FUNCTION_BLOCK FB_Lifetime_Predictor
  VAR_INPUT
    VI_Runtime_Hours : UDINT;
    VI_Start_Count : UDINT;
    VI_Nominal_Life : UDINT := 10000;
  END_VAR
  VAR_OUTPUT
    VO_Remaining_Percent : BYTE;
    VO_Maintenance_Req : BOOL;
  END_VAR

            // Упрощенная модель износа
IF VI_Nominal_Life > 0 THEN
    VO_Remaining_Percent := TO_BYTE(100 - (VI_Runtime_Hours * 100 / VI_Nominal_Life));
ELSE
    VO_Remaining_Percent := 0;
END_IF;

VO_Maintenance_Req := (VO_Remaining_Percent < 10);
          
END_FUNCTION_BLOCK

FUNCTION_BLOCK FB_System_Alarm_Orchestrator
  VAR_INPUT
    VI_First_Fault_Active : BOOL;
    VI_First_Fault_Type : INT;
    VI_First_Fault_Source : INT;
  END_VAR
  VAR
    fbAlarmManager : FB_Alarm_Manager;
  END_VAR

            // ==============================================================================
// System alarm orchestrator helper
//
// Internal helper for PRG_System.
// Owns FB_Alarm_Manager call and alarm output projection.
// ==============================================================================



fbAlarmManager(
    VI_System_Time_MS := GVL_STATUS.G_System_Time_MS,
    VI_IsActivePLC := GVL_STATUS.G_Is_Active_PLC,
    VI_Gas_Alarm := GVL_HEALTH_BRIDGE.G_Gas_Detected OR GVL_HEALTH_BRIDGE.G_CO_Alarm_Level,
    VI_Fire_Alarm := GVL_HEALTH_BRIDGE.G_Smoke_Detected,
    VI_Flood_Alarm := GVL_HEALTH_BRIDGE.G_Leak_Detected,
    VI_Security_Alarm := GVL_ALARM.G_Security_Alarm,
    VI_First_Fault_Active := VI_First_Fault_Active,
    VI_First_Fault_Type := VI_First_Fault_Type,
    VI_First_Fault_Source := VI_First_Fault_Source,
    VI_Boiler_Errors := GVL_STATE.G_Boiler_Error,
    VI_Security_Msg := GVL_STATUS.G_Security_Status_Msg,
    VI_Acknowledge_All := GVL_CONFIG.G_HMI_Ack_Alarms OR GVL_COMMAND.G_Reset_Errors,
    VI_Mute_Siren := GVL_CONFIG.G_HMI_Mute_Alarm,
    VIO_Next_Alarm_ID := GVL_ALARM.G_Next_Alarm_ID,
    VO_Global_Critical => GVL_ALARM.G_Global_Critical,
    VO_Global_Warning => GVL_ALARM.G_Global_Warning,
    VO_Siren_Active => GVL_ALARM.G_Global_Siren,
    VO_Active_Count => GVL_ALARM.G_Active_Alarm_Count,
    VO_Unacked_Count => GVL_ALARM.G_Unacked_Alarm_Count,
    VO_Event_Pulse => GVL_STATUS.G_Diagnostics.Alarm_Event_Pulse,
    VO_Event_Code => GVL_STATUS.G_Diagnostics.Alarm_Event_Code,
    VO_Event_Value => GVL_STATUS.G_Diagnostics.Alarm_Event_Value,
    VO_Alarm_List => GVL_ALARM.G_Alarm_List
);

// >>> BULK_SYNC_ANCHOR: FB_System_Alarm_Orchestrator <<<
          
END_FUNCTION_BLOCK

FUNCTION_BLOCK FB_Heating_Runtime_Timeline_Observer
  VAR_INPUT
    VI_Enable : BOOL;
    VI_Frame : ST_Heating_Runtime_Execution_Frame;
  END_VAR
  VAR_IN_OUT
    VIO_Timeline : ST_Heating_Runtime_Execution_Timeline;
  END_VAR
  VAR
    L_Index : UINT;
  END_VAR

            // ==============================================================================
// Heating runtime timeline observer
// Read-only deterministic execution timeline layer.
// ==============================================================================



IF NOT VI_Enable THEN
    RETURN;
END_IF;

// ======================================================
// SAFE INDEX NORMALIZATION
// ======================================================
IF (VIO_Timeline.Write_Index < 1) OR
   (VIO_Timeline.Write_Index >= 64) THEN

    L_Index := 1;

    IF VIO_Timeline.Write_Index >= 64 THEN
        VIO_Timeline.Timeline_Overflow := TRUE;
    END_IF;

ELSE
    L_Index := VIO_Timeline.Write_Index + 1;
END_IF;

// ======================================================
// FRAME STORAGE
// ======================================================
VIO_Timeline.Frames[L_Index] := VI_Frame;
VIO_Timeline.Write_Index := L_Index;

IF VIO_Timeline.Frame_Count < 64 THEN
    VIO_Timeline.Frame_Count :=
        VIO_Timeline.Frame_Count + 1;
END_IF;

// ======================================================
// TELEMETRY UPDATE
// ======================================================
VIO_Timeline.Sequencing_Valid :=
    VI_Frame.Sequencing_Valid;

VIO_Timeline.Ownership_Valid :=
    VI_Frame.Ownership_Valid;

VIO_Timeline.Synchronization_Valid :=
    VI_Frame.Synchronization_Valid;

VIO_Timeline.Runtime_Jitter_Detected :=
    VI_Frame.Runtime_Jitter_Detected;

VIO_Timeline.Runtime_Latency_Detected :=
    VI_Frame.Runtime_Latency_Detected;

VIO_Timeline.Runtime_Degraded :=
    VI_Frame.Runtime_Degraded;

VIO_Timeline.Status_Code := VI_Frame.Status_Code;
VIO_Timeline.Status_Text := VI_Frame.Status_Text;

// >>> BULK_SYNC_ANCHOR: FB_Heating_Runtime_Timeline_Observer <<<
          
END_FUNCTION_BLOCK

FUNCTION_BLOCK FB_Behavior_Adapt
  VAR_INPUT
    iScenario : E_System_Reason_Code;
    iSuccess : BOOL;
    iMeasuredValue : REAL;
    iZone : INT;
    iConfidence : REAL;
  END_VAR
  VAR
    L_Stats : ST_Scenario_Stats;
    L_Zone : ST_Zone_Adapt_State;
    L_Adjustment : REAL;
    L_Decay : REAL;
    idx : INT;
  END_VAR

            IF NOT GVL_BEHAVIOR_ADAPT.G_Adapt_Enabled THEN RETURN; END_IF;

idx := USINT_TO_INT(iScenario);

L_Stats := GVL_BEHAVIOR_ADAPT.G_Scenario_Stats[idx];
L_Stats.Activations := L_Stats.Activations + 1;

IF iSuccess THEN
    L_Stats.Success_Count := L_Stats.Success_Count + 1;
ELSE
    L_Stats.Failure_Count := L_Stats.Failure_Count + 1;
END_IF;

IF L_Stats.Activations > 0 THEN
    L_Stats.Success_Rate := UDINT_TO_REAL(L_Stats.Success_Count) / UDINT_TO_REAL(L_Stats.Activations);
END_IF;

IF (iScenario = REASON_SCENARIO_VENT_BOOST) AND (iZone >= 1) AND (iZone <= GVL_CONSTANTS.C_MAX_ZONES) THEN

    L_Zone := GVL_BEHAVIOR_ADAPT.G_VentBoost_Zone_Adapt[iZone];

    IF L_Zone.Zone_Weight = 0.0 THEN
        L_Zone.Zone_Weight := GVL_BEHAVIOR_ADAPT.G_Adapt_Default_Zone_Weight;
    END_IF;

    L_Decay := GVL_BEHAVIOR_ADAPT.G_Decay_Factor;
    L_Zone.Zone_Weight := L_Zone.Zone_Weight * L_Decay;
    L_Zone.Confidence := L_Zone.Confidence * L_Decay;

    L_Zone.Activations := L_Zone.Activations + 1;

    IF iSuccess THEN
        L_Zone.Success_Count := L_Zone.Success_Count + 1;
    ELSE
        L_Zone.Failure_Count := L_Zone.Failure_Count + 1;
    END_IF;

    IF L_Zone.Activations > 0 THEN
        L_Zone.Success_Rate := UDINT_TO_REAL(L_Zone.Success_Count) / UDINT_TO_REAL(L_Zone.Activations);
    END_IF;

    IF iConfidence >= GVL_BEHAVIOR_ADAPT.G_Adapt_Min_Confidence THEN
        L_Zone.Confidence := L_Zone.Confidence +
            (iConfidence - L_Zone.Confidence) * GVL_BEHAVIOR_ADAPT.G_Confidence_Learning_Rate;
    END_IF;

    IF (GVL_BEHAVIOR_ADAPT.G_Adapt_Update_Threshold > 0) AND
       ((L_Zone.Activations MOD INT_TO_UDINT(GVL_BEHAVIOR_ADAPT.G_Adapt_Update_Threshold)) = 0) THEN

        L_Adjustment :=
            (L_Zone.Success_Rate - 0.5)
            * GVL_BEHAVIOR_ADAPT.G_Adapt_Learning_Rate
            * L_Zone.Confidence;

        L_Zone.Zone_Weight := LIMIT(0.5, L_Zone.Zone_Weight + L_Adjustment, 2.0);

    END_IF;

    L_Zone.Last_Update_MS := GVL_TIME_SERVICE.G_Now_MS;

    GVL_BEHAVIOR_ADAPT.G_VentBoost_Zone_Adapt[iZone] := L_Zone;

END_IF;

GVL_BEHAVIOR_ADAPT.G_Scenario_Stats[idx] := L_Stats;
          
END_FUNCTION_BLOCK

FUNCTION_BLOCK FB_Heating_Optimizer
  VAR
    L_i : INT;
    L_Load : REAL;
    L_Total_Demand : REAL;
  END_VAR

            // ==============================================================================
// Ownership note
// ------------------------------------------------------------------------------
// This block calculates optimization diagnostics only.
// It does NOT modify thermal demand.
//
// Thermal demand ownership remains in:
// FB_Heating_Thermal_Model.
// ==============================================================================

L_Total_Demand := 0.0;

// Aggregate thermal load estimate.
FOR L_i := 1 TO GVL_CONSTANTS.C_MAX_ZONES DO
    L_Total_Demand := L_Total_Demand + ABS(GVL_HEATING_POLICY.G_Zone_Thermal_Demand[L_i]);
END_FOR;

GVL_HEATING_POLICY.G_Optimization_Load_Index := L_Total_Demand;
GVL_HEATING_POLICY.G_Optimization_Energy_Saving_Active := FALSE;

// Zone optimization diagnostics.
FOR L_i := 1 TO GVL_CONSTANTS.C_MAX_ZONES DO

    IF L_Total_Demand > 0.01 THEN
        L_Load := ABS(GVL_HEATING_POLICY.G_Zone_Thermal_Demand[L_i]) / L_Total_Demand;
    ELSE
        L_Load := 0.0;
    END_IF;

    GVL_HEATING_POLICY.G_Zone_Optimization_Score[L_i] :=
        L_Load +
        ((1.0 - GVL_HEATING_POLICY.G_Zone_Thermal_Model_Confidence[L_i]) * 0.2);

    // Advisory energy-saving indication only.
    IF L_Total_Demand > 5.0 THEN
        GVL_HEATING_POLICY.G_Optimization_Energy_Saving_Active := TRUE;
    END_IF;

END_FOR;
          
END_FUNCTION_BLOCK

FUNCTION_BLOCK FB_System_Timebase
  VAR
    L_Time_Diff : UDINT;
  END_VAR

            // ==============================================================================
// System timebase helper
//
// Internal helper for PRG_System.
// Owns PLC runtime clock projection into GVL_STATUS:
// - monotonic system milliseconds
// - time-of-day milliseconds
// - day of week / day of year rollover
// - TOD representation
// ==============================================================================



GVL_STATUS.G_System_Time_MS := TIME_TO_UDINT(TIME());

L_Time_Diff := SEL(
    GVL_STATUS.G_System_Time_MS >= GVL_STATUS.G_Last_System_Time_MS,
    GVL_STATUS.G_System_Time_MS - GVL_STATUS.G_Last_System_Time_MS,
    (4294967295 - GVL_STATUS.G_Last_System_Time_MS) + GVL_STATUS.G_System_Time_MS + 1
);

GVL_STATUS.G_Time_Of_Day_MS := (GVL_STATUS.G_Time_Of_Day_MS + L_Time_Diff) MOD 86400000;

IF GVL_STATUS.G_Time_Of_Day_MS < L_Time_Diff THEN
    GVL_STATUS.G_Current_Day := (GVL_STATUS.G_Current_Day MOD 7) + 1;
    GVL_STATUS.G_Day_Of_Year := (GVL_STATUS.G_Day_Of_Year MOD 365) + 1;
END_IF;

GVL_STATUS.G_Last_System_Time_MS := GVL_STATUS.G_System_Time_MS;
GVL_STATUS.G_Current_TOD := UDINT_TO_TOD(GVL_STATUS.G_Time_Of_Day_MS);

// >>> BULK_SYNC_ANCHOR: FB_System_Timebase <<<
          
END_FUNCTION_BLOCK

FUNCTION_BLOCK FB_Redundancy_Manager
  VAR_INPUT
    VI_System_Time_MS : UDINT;
    VI_Local_PLC_ID : BYTE;
    VI_Remote_Pulse : BOOL;
    VI_Remote_Is_Active : BOOL;
    VI_Gateway_Ping_OK : BOOL;
    VI_Remote_State : ST_System_State_Snapshot;
    VI_Local_State : ST_System_State_Snapshot;
  END_VAR
  VAR_OUTPUT
    VO_Local_Role : E_PLC_ROLE;
    VO_Local_Pulse : BOOL;
    VO_Sync_Data_Req : BOOL;
    VO_Status_Msg : STRING(200);
    VO_Synced_State : ST_System_State_Snapshot;
    VO_State_Updated : BOOL;
  END_VAR
  VAR
    L_Heartbeat : FB_PLC_Heartbeat;
    L_Pulse_Timer : FB_System_Timer;
    L_Pulse_State : BOOL;
    L_Prev_Role : E_PLC_ROLE;
    L_State_Replicator : FB_State_Replication;
  END_VAR

            // 1. Генерация собственного пульса (меандр 100 мс)
L_Pulse_Timer(IN := NOT L_Pulse_Timer.Q, PT := T#100ms, VI_System_Time_MS := VI_System_Time_MS);
IF L_Pulse_Timer.Q THEN
    L_Pulse_State := NOT L_Pulse_State;
END_IF;
VO_Local_Pulse := L_Pulse_State;

// 2. Определение роли через Heartbeat
L_Heartbeat(
    VI_Local_ID := VI_Local_PLC_ID,
    VI_System_Time := VI_System_Time_MS,
    VI_Remote_Pulse := VI_Remote_Pulse,
    VI_Remote_Is_Active := VI_Remote_Is_Active,
    VI_Gateway_Ping_OK := VI_Gateway_Ping_OK
);

IF L_Heartbeat.VO_Is_Active THEN
    VO_Local_Role := E_PLC_ROLE.ROLE_ACTIVE;
    VO_Status_Msg := 'ПЛК АКТИВЕН (ВЕДУЩИЙ)';
ELSE
    VO_Local_Role := E_PLC_ROLE.ROLE_STANDBY;
    VO_Status_Msg := 'ПЛК В РЕЗЕРВЕ (ВЕДОМЫЙ)';
END_IF;

// 3. Запрос на синхронизацию при переходе в ACTIVE
IF VO_Local_Role = E_PLC_ROLE.ROLE_ACTIVE AND L_Prev_Role = E_PLC_ROLE.ROLE_STANDBY THEN
    VO_Sync_Data_Req := TRUE;
ELSE
    VO_Sync_Data_Req := FALSE;
END_IF;

L_State_Replicator(
    VI_Local_Role := VO_Local_Role,
    VI_Sync_Req := VO_Sync_Data_Req,
    VI_Local_State := VI_Local_State,
    VI_Remote_State := VI_Remote_State,
    VI_System_Time_MS := VI_System_Time_MS
);
VO_Synced_State := L_State_Replicator.VO_Synced_State;
VO_State_Updated := L_State_Replicator.VO_State_Updated;

L_Prev_Role := VO_Local_Role;
// >>> BULK_SYNC_ANCHOR: FB_Redundancy_Manager <<<
          
END_FUNCTION_BLOCK

FUNCTION_BLOCK FB_System_Redundancy_Orchestrator
  VAR_IN_OUT
    VIO_Local_State : ST_System_State_Snapshot;
    VIO_Remote_State : ST_System_State_Snapshot;
  END_VAR
  VAR
    fbRedundancy : FB_Redundancy_Manager;
  END_VAR

            // ==============================================================================
// System redundancy orchestrator helper
//
// Internal helper for PRG_System.
// Owns PLC role calculation, heartbeat output projection, and synced-state apply.
// ==============================================================================



// Build local state snapshot for replication.
VIO_Local_State.System_Time_MS := GVL_STATUS.G_System_Time_MS;
VIO_Local_State.Current_Scenario := GVL_STATUS.G_Current_Scenario;
VIO_Local_State.Security_Armed := GVL_ALARM.G_Security_Armed;
VIO_Local_State.Active_Alarms := GVL_ALARM.G_Active_Alarm_Count;
VIO_Local_State.Zone_Valves := GVL_STATE.G_Zone_Valves;
VIO_Local_State.Manifold_Pumps := GVL_STATE.G_Manifold_Pumps;
VIO_Local_State.Lighting_States := GVL_STATE.G_Lighting_Levels;
VIO_Local_State.Blinds_Positions := GVL_STATE.G_Blinds_Positions;
VIO_Local_State.Socket_States := GVL_STATE.G_Socket_States;
VIO_Local_State.Gas_Valve_Closed := GVL_COMMAND.G_Gas_Valve_Close;
VIO_Local_State.Water_Valves_Closed := GVL_COMMAND.G_Close_Valve_36;
VIO_Local_State.Version := VIO_Local_State.Version + 1;

fbRedundancy(
    VI_System_Time_MS := GVL_STATUS.G_System_Time_MS,
    VI_Local_PLC_ID := GVL_STATUS.G_PLC_ID,
    VI_Remote_Pulse := GVL_IO.DI_Partner_Pulse,
    VI_Remote_Is_Active := GVL_IO.DI_Partner_Active,
    VI_Gateway_Ping_OK := GVL_GATEWAY.G_Gateway_Ping_OK,
    VI_Local_State := VIO_Local_State,
    VI_Remote_State := VIO_Remote_State
);

GVL_STATUS.G_Is_Active_PLC := (fbRedundancy.VO_Local_Role = E_PLC_ROLE.ROLE_ACTIVE);
GVL_IO.DO_Heartbeat_Pulse := fbRedundancy.VO_Local_Pulse;
GVL_IO.DO_Active_Status := GVL_STATUS.G_Is_Active_PLC;

IF fbRedundancy.VO_State_Updated THEN
    GVL_STATUS.G_Current_Scenario := fbRedundancy.VO_Synced_State.Current_Scenario;
    GVL_ALARM.G_Security_Armed := fbRedundancy.VO_Synced_State.Security_Armed;
    GVL_STATE.G_Zone_Valves := fbRedundancy.VO_Synced_State.Zone_Valves;
    GVL_STATE.G_Manifold_Pumps := fbRedundancy.VO_Synced_State.Manifold_Pumps;
    GVL_STATE.G_Lighting_Levels := fbRedundancy.VO_Synced_State.Lighting_States;
    GVL_STATE.G_Blinds_Positions := fbRedundancy.VO_Synced_State.Blinds_Positions;
    GVL_STATE.G_Socket_States := fbRedundancy.VO_Synced_State.Socket_States;
    GVL_COMMAND.G_Gas_Valve_Close := fbRedundancy.VO_Synced_State.Gas_Valve_Closed;
    GVL_COMMAND.G_Close_Valve_36 := fbRedundancy.VO_Synced_State.Water_Valves_Closed;
    VIO_Local_State.Version := fbRedundancy.VO_Synced_State.Version;
END_IF;

// >>> BULK_SYNC_ANCHOR: FB_System_Redundancy_Orchestrator <<<
          
END_FUNCTION_BLOCK

FUNCTION_BLOCK FB_Heating_Boiler_Control
  VAR_INPUT
    VI_System_Time_MS : UDINT;
    VI_IsActivePLC : BOOL;
    VI_DHW_Heating_Demand : BOOL;
    VI_DHW_Target_Temp : REAL;
    VI_Target_Supply_Temp : REAL;
    VI_Freeze_Mode_Active : BOOL;
    VI_Policy_Degraded : BOOL;
    VI_Manifold_Pumps : ARRAY[1..GVL_CONSTANTS.C_MAX_MANIFOLDS] OF BOOL;
    VI_Manifold_Valves : ARRAY[1..GVL_CONSTANTS.C_MAX_MANIFOLDS] OF REAL;
    VI_Boiler_Flame_Status : ARRAY[1..GVL_CONSTANTS.C_MAX_BOILERS] OF BOOL;
    VI_Boiler_Error_Status : ARRAY[1..GVL_CONSTANTS.C_MAX_BOILERS] OF BOOL;
    VI_Boiler_OT_Online : ARRAY[1..GVL_CONSTANTS.C_MAX_BOILERS] OF BOOL;
  END_VAR
  VAR_OUTPUT
    VO_Boiler_OT_Enable : ARRAY[1..GVL_CONSTANTS.C_MAX_BOILERS] OF BOOL;
    VO_Boiler_OT_Setpoint : ARRAY[1..GVL_CONSTANTS.C_MAX_BOILERS] OF REAL;
    VO_Boiler_Status : ARRAY[1..GVL_CONSTANTS.C_MAX_BOILERS] OF ST_Boiler_Status;
    VO_Any_Subsystem_Degraded : BOOL;
    VO_Lead_Boiler : BYTE;
    VO_Demand_Power : REAL;
  END_VAR
  VAR_IN_OUT
    VI_Boiler_Modulation : ARRAY[1..GVL_CONSTANTS.C_MAX_BOILERS] OF REAL;
  END_VAR
  VAR
    L_i : INT;
    L_Delta_MS : UDINT;
    L_Last_Scan_Time : UDINT;
    L_Scan_Time_Init : BOOL := FALSE;
    L_Boiler_Request_Enable : ARRAY[1..GVL_CONSTANTS.C_MAX_BOILERS] OF BOOL;
    L_Boiler_Request_Setpoint : ARRAY[1..GVL_CONSTANTS.C_MAX_BOILERS] OF REAL;
    L_Boiler_OT_Command_Valid : ARRAY[1..GVL_CONSTANTS.C_MAX_BOILERS] OF BOOL;
    L_Transport_Degraded : BOOL;
    L_Available_Count : UINT;
    L_Active_Count : UINT;
    L_Any_Transport_Degraded : BOOL;
    L_Any_Ignition_Timeout : BOOL;
    L_Any_Flame : BOOL;
    L_Boiler_Life : ARRAY[1..GVL_CONSTANTS.C_MAX_BOILERS] OF FB_Lifetime_Predictor;
    fbBoilerCascade : FB_Boiler_Cascade_Manager;
    fbBoilerOpenTherm : FB_Boiler_OpenTherm_Interface;
  END_VAR

            // ==============================================================================
// Heating boiler control helper
// ==============================================================================



VO_Any_Subsystem_Degraded := FALSE;
VO_Demand_Power := 0.0;

L_Available_Count := 0;
L_Active_Count := 0;
L_Any_Transport_Degraded := FALSE;
L_Any_Ignition_Timeout := FALSE;
L_Any_Flame := FALSE;

FOR L_i := 1 TO GVL_CONSTANTS.C_MAX_MANIFOLDS DO
    IF VI_Manifold_Pumps[L_i] THEN
        VO_Demand_Power := VO_Demand_Power + VI_Manifold_Valves[L_i];
    END_IF;
END_FOR;

IF VI_Freeze_Mode_Active AND VO_Demand_Power < 20.0 THEN
    VO_Demand_Power := 20.0;
END_IF;

IF VI_Policy_Degraded THEN
    IF VO_Demand_Power > 60.0 THEN
        VO_Demand_Power := 60.0;
    END_IF;
END_IF;

fbBoilerCascade(
    VI_Enable := VI_IsActivePLC AND ((VO_Demand_Power > GVL_CONSTANTS.C_BOILER_CASCADE_MIN_DEMAND) OR VI_Freeze_Mode_Active OR VI_DHW_Heating_Demand),
    VI_System_Time_MS := VI_System_Time_MS,
    VI_Boiler_Stop := FALSE,
    VI_DHW_Heating_Demand := VI_DHW_Heating_Demand,
    VI_DHW_Target_Temp := VI_DHW_Target_Temp,
    VI_Target_Supply_Temp := VI_Target_Supply_Temp,
    VI_Demand_Power := VO_Demand_Power,
    VI_Boiler_Flame_Status := VI_Boiler_Flame_Status,
    VI_Boiler_Error_Status := VI_Boiler_Error_Status,
    VI_Boiler_OT_Online := VI_Boiler_OT_Online,
    VI_Boiler_Modulation := VI_Boiler_Modulation,
    VO_Boiler_Enable => L_Boiler_Request_Enable,
    VO_Boiler_Setpoint => L_Boiler_Request_Setpoint,
    VO_Lead_Boiler => VO_Lead_Boiler
);

FOR L_i := 1 TO GVL_CONSTANTS.C_MAX_BOILERS DO
    IF L_Boiler_Request_Enable[L_i] THEN
        L_Boiler_Request_Setpoint[L_i] := LIMIT(
            GVL_CONSTANTS.C_BOILER_SETPOINT_MIN,
            L_Boiler_Request_Setpoint[L_i],
            80.0
        );
    END_IF;
END_FOR;

FOR L_i := 1 TO GVL_CONSTANTS.C_MAX_BOILERS DO
    IF NOT VI_Boiler_OT_Online[L_i] OR VI_Boiler_Error_Status[L_i] THEN
        L_Boiler_Request_Enable[L_i] := FALSE;
        L_Boiler_Request_Setpoint[L_i] := 0.0;
    END_IF;
END_FOR;

fbBoilerOpenTherm(
    VI_Enable := L_Boiler_Request_Enable,
    VI_Setpoint := L_Boiler_Request_Setpoint,
    VI_OT_Online := VI_Boiler_OT_Online,
    VI_OT_Error := VI_Boiler_Error_Status,
    VO_OT_Enable => VO_Boiler_OT_Enable,
    VO_OT_Setpoint => VO_Boiler_OT_Setpoint,
    VO_OT_Command_Valid => L_Boiler_OT_Command_Valid
);

FOR L_i := 1 TO GVL_CONSTANTS.C_MAX_BOILERS DO

    L_Transport_Degraded :=
        L_Boiler_Request_Enable[L_i] AND
        (
            NOT L_Boiler_OT_Command_Valid[L_i] OR
            NOT VI_Boiler_OT_Online[L_i] OR
            VI_Boiler_Error_Status[L_i]
        );

    VO_Boiler_Status[L_i].OT_Online := VI_Boiler_OT_Online[L_i];
    VO_Boiler_Status[L_i].OT_Command_Valid := L_Boiler_OT_Command_Valid[L_i];
    VO_Boiler_Status[L_i].OT_Transport_Degraded := L_Transport_Degraded;
    VO_Boiler_Status[L_i].OT_Adapter_Error :=
        GVL_OPENTHERM_ADAPTER.G_Status[L_i].Adapter_Error;

    VO_Boiler_Status[L_i].Active := L_Boiler_Request_Enable[L_i];
    VO_Boiler_Status[L_i].Running := VI_Boiler_Flame_Status[L_i];
    VO_Boiler_Status[L_i].Warning := L_Transport_Degraded;
    VO_Boiler_Status[L_i].Error := VI_Boiler_Error_Status[L_i];

    VO_Boiler_Status[L_i].Available :=
        VI_Boiler_OT_Online[L_i] AND
        NOT VI_Boiler_Error_Status[L_i] AND
        NOT L_Transport_Degraded;

    VO_Boiler_Status[L_i].Selected_By_Cascade :=
        L_Boiler_Request_Enable[L_i];

    VO_Boiler_Status[L_i].Transport_Missing :=
        NOT VI_Boiler_OT_Online[L_i];

    VO_Boiler_Status[L_i].Flame_Missing :=
        L_Boiler_Request_Enable[L_i] AND
        NOT VI_Boiler_Flame_Status[L_i] AND
        NOT L_Transport_Degraded;

    VO_Boiler_Status[L_i].Ignition_Timeout :=
        VO_Boiler_Status[L_i].Flame_Missing AND
        (GVL_STATE.G_Boiler_OT_Command_Age_MS[L_i] > 30000);

    VO_Boiler_Status[L_i].Degraded :=
        L_Transport_Degraded OR
        VO_Boiler_Status[L_i].Ignition_Timeout;

    // ======================================================
    // CASCADE AGGREGATION
    // ======================================================
    IF VO_Boiler_Status[L_i].Available THEN
        L_Available_Count := L_Available_Count + 1;
    END_IF;

    IF VO_Boiler_Status[L_i].Selected_By_Cascade THEN
        L_Active_Count := L_Active_Count + 1;
    END_IF;

    IF VI_Boiler_Flame_Status[L_i] THEN
        L_Any_Flame := TRUE;
    END_IF;

    IF L_Transport_Degraded THEN
        L_Any_Transport_Degraded := TRUE;
    END_IF;

    IF VO_Boiler_Status[L_i].Ignition_Timeout THEN
        L_Any_Ignition_Timeout := TRUE;
    END_IF;

    IF VO_Boiler_Status[L_i].Degraded THEN
        VO_Any_Subsystem_Degraded := TRUE;
    END_IF;

END_FOR;

// ======================================================
// GLOBAL CASCADE SEMANTIC STATE
// ======================================================
GVL_STATE.G_Heating_Cascade_Active_Boilers := L_Active_Count;
GVL_STATE.G_Heating_Cascade_Available_Boilers := L_Available_Count;

GVL_STATE.G_Heating_Cascade_Available :=
    (L_Available_Count > 0);

GVL_STATE.G_Heating_Cascade_Partial_Capacity :=
    (L_Available_Count > 0) AND
    (L_Available_Count < GVL_CONSTANTS.C_MAX_BOILERS);

GVL_STATE.G_Heating_Cascade_Transport_Degraded :=
    L_Any_Transport_Degraded;

GVL_STATE.G_Heating_Cascade_Ignition_Timeout :=
    L_Any_Ignition_Timeout;

GVL_STATE.G_Heating_Cascade_No_Flame :=
    (L_Active_Count > 0) AND
    NOT L_Any_Flame;

GVL_STATE.G_Heating_Cascade_Degraded :=
    GVL_STATE.G_Heating_Cascade_Transport_Degraded OR
    GVL_STATE.G_Heating_Cascade_Ignition_Timeout OR
    GVL_STATE.G_Heating_Cascade_Partial_Capacity;
          
END_FUNCTION_BLOCK

FUNCTION_BLOCK FB_System_Timer
  VAR_INPUT
    IN : BOOL;
    PT : TIME;
    VI_System_Time_MS : UDINT;
  END_VAR
  VAR_OUTPUT
    Q : BOOL;
    ET : TIME;
  END_VAR
  VAR
    L_Start_Time : UDINT;
    L_Running : BOOL;
  END_VAR

            // ==============================================================================
// Блок таймера, привязанный к системному времени (System Timer)
// Назначение:
// - Замена стандартного TON для обеспечения точной выдержки времени,
//   независимой от времени цикла ПЛК, с использованием единого системного времени.
// ==============================================================================



IF IN THEN
    IF NOT L_Running THEN
        L_Start_Time := VI_System_Time_MS;
        L_Running := TRUE;
        ET := T#0s;
        Q := FALSE;
    ELSE
        // Обработка переполнения UDINT (примерно 49 дней)
        ET := TO_TIME((SEL(VI_System_Time_MS >= L_Start_Time, VI_System_Time_MS - L_Start_Time, (4294967295 - L_Start_Time) + VI_System_Time_MS + 1)));
        
        IF ET >= PT THEN
            Q := TRUE;
            ET := PT;
        ELSE
            Q := FALSE;
        END_IF;
    END_IF;
ELSE
    L_Running := FALSE;
    ET := T#0s;
    Q := FALSE;
END_IF;
// >>> BULK_SYNC_ANCHOR: FB_System_Timer <<<
          
END_FUNCTION_BLOCK

FUNCTION_BLOCK FB_Heating_Runtime_Supervisory_Publication_Adapter
  VAR_INPUT
    VI_Enable : BOOL;
    VI_Predictive_State : ST_Heating_Runtime_Predictive_State;
    VI_Causality_Node : ST_Heating_Runtime_Causality_Node;
    VI_Causality_Edge : ST_Heating_Runtime_Causality_Edge;
    VI_Blackbox_Event : ST_Heating_Runtime_Blackbox_Event;
    VI_Anomaly : ST_Heating_Runtime_Anomaly;
  END_VAR

            IF NOT VI_Enable THEN
    RETURN;
END_IF;

GVL_Heating_Runtime_Supervisory_Publication.G_Publication.Supervisory_Visible := TRUE;
GVL_Heating_Runtime_Supervisory_Publication.G_Publication.Predictive_State := VI_Predictive_State;
GVL_Heating_Runtime_Supervisory_Publication.G_Publication.Source_Instability_Attention := VI_Predictive_State.Source_Instability_Attention;
GVL_Heating_Runtime_Supervisory_Publication.G_Publication.Source_Oscillation_Trend_Visible := VI_Predictive_State.Source_Oscillation_Trend_Visible;
GVL_Heating_Runtime_Supervisory_Publication.G_Publication.Runtime_Degraded := VI_Anomaly.Runtime_Degraded;
GVL_Heating_Runtime_Supervisory_Publication.G_Publication.Runtime_Fault := VI_Anomaly.Critical_Anomaly;
GVL_Heating_Runtime_Supervisory_Publication.G_Publication.Explainability_Degraded := VI_Anomaly.Explainability_Degraded;
GVL_Heating_Runtime_Supervisory_Publication.G_Publication.Diagnostics_Degraded := VI_Anomaly.Diagnostics_Degraded;
GVL_Heating_Runtime_Supervisory_Publication.G_Publication.Causality_Active := VI_Causality_Node.Node_Active;
GVL_Heating_Runtime_Supervisory_Publication.G_Publication.Propagation_Detected := VI_Causality_Edge.Propagation_Detected;
GVL_Heating_Runtime_Supervisory_Publication.G_Publication.Reconstruction_Visible := VI_Blackbox_Event.Event_Active;
GVL_Heating_Runtime_Supervisory_Publication.G_Publication.Status_Code := VI_Predictive_State.Status_Code;
GVL_Heating_Runtime_Supervisory_Publication.G_Publication.Status_Text := VI_Predictive_State.Status_Text;
          
END_FUNCTION_BLOCK

FUNCTION_BLOCK FB_Heating_Runtime_Stability_Model
  VAR_INPUT
    VI_Enable : BOOL;
    VI_Runtime_Degraded : BOOL;
    VI_Runtime_Critical : BOOL;
  END_VAR
  VAR_OUTPUT
    VO_Runtime_Stable : BOOL;
    VO_Stability_Score : UINT;
    VO_Status_Code : UINT;
    VO_Status_Text : STRING(128);
  END_VAR

            // ==============================================================================
// Heating runtime stability model
// Read-only predictive runtime stability layer.
// ==============================================================================



VO_Runtime_Stable := FALSE;
VO_Stability_Score := 0;

VO_Status_Code := 0;
VO_Status_Text := 'Heating runtime stability model disabled';

IF NOT VI_Enable THEN
    RETURN;
END_IF;

IF VI_Runtime_Critical THEN
    VO_Runtime_Stable := FALSE;
    VO_Stability_Score := 0;

    VO_Status_Code := 900;
    VO_Status_Text := 'Heating runtime critically unstable';

ELSIF VI_Runtime_Degraded THEN
    VO_Runtime_Stable := FALSE;
    VO_Stability_Score := 50;

    VO_Status_Code := 200;
    VO_Status_Text := 'Heating runtime degraded stability';

ELSE
    VO_Runtime_Stable := TRUE;
    VO_Stability_Score := 100;

    VO_Status_Code := 1;
    VO_Status_Text := 'Heating runtime stable';
END_IF;

// >>> BULK_SYNC_ANCHOR: FB_Heating_Runtime_Stability_Model <<<
          
END_FUNCTION_BLOCK

FUNCTION_BLOCK FB_Water_Physical_Runtime
  VAR_INPUT
    VI_Enable : BOOL;
    VI_System_Time_MS : UDINT;
  END_VAR
  VAR
    L_i : INT;
    L_Output : ST_Water_Output_Projection_State;
    L_Feedback : ST_Water_Valve_Feedback_State;
    L_Convergence : ST_Water_Physical_Convergence_State;
    L_Diagnostics : ST_Water_Actuator_Diagnostics_State;
    L_Any_Convergence_Degraded : BOOL;
    L_Any_Diagnostics_Degraded : BOOL;
    L_Any_Escalation : BOOL;
  END_VAR

            IF NOT VI_Enable THEN
    GVL_Water_Physical_Runtime.G_Runtime_Valid := FALSE;
    RETURN;
END_IF;

FOR L_i := 1 TO GVL_CONSTANTS.C_MAX_FLOOD_SENSORS DO
    L_Output := GVL_Water_Output_Projection.G_Output_Projection_State[L_i];
    L_Feedback := GVL_Water_Valve_Feedback.G_Valve_Feedback_State[L_i];

    L_Convergence.Runtime_Valid := TRUE;
    L_Convergence.Runtime_System_Time_MS := VI_System_Time_MS;
    L_Convergence.Sensor_Id := TO_UINT(L_i);
    L_Convergence.Projection_Active := L_Output.Projection_Allowed;
    L_Convergence.Physical_Open_Confirmed := L_Feedback.Confirmed_Open;
    L_Convergence.Physical_Closed_Confirmed := L_Feedback.Confirmed_Closed;
    L_Convergence.Physical_State_Confirmed := L_Feedback.Confirmed_Open OR L_Feedback.Confirmed_Closed;

    IF L_Feedback.Feedback_Available THEN
        IF L_Output.Expected_Closed AND NOT L_Feedback.Confirmed_Closed THEN
            L_Convergence.Projection_Mismatch := TRUE;
            L_Convergence.Physical_Mismatch := TRUE;
        END_IF;

        IF NOT L_Convergence.Projection_Mismatch AND NOT L_Feedback.Feedback_Timeout THEN
            L_Convergence.Runtime_Converged := TRUE;
        END_IF;
    ELSE
        L_Convergence.Runtime_Mismatch := FALSE;
    END_IF;

    IF L_Convergence.Projection_Mismatch OR L_Feedback.Feedback_Conflict THEN
        L_Convergence.Convergence_Degraded := TRUE;
        L_Convergence.Escalation_Required := TRUE;
        L_Convergence.Status_Code := 2;
        L_Convergence.Status_Text := 'Physical convergence mismatch detected';
    ELSIF L_Convergence.Runtime_Converged THEN
        L_Convergence.Status_Code := 1;
        L_Convergence.Status_Text := 'Physical runtime converged';
    ELSE
        L_Convergence.Status_Code := 0;
        L_Convergence.Status_Text := 'Physical convergence observe-only';
    END_IF;

    L_Diagnostics.Runtime_Valid := TRUE;
    L_Diagnostics.Runtime_System_Time_MS := VI_System_Time_MS;
    L_Diagnostics.Valve_Group_Id := L_Output.Valve_Group_Id;
    L_Diagnostics.Travel_Active := L_Output.Projection_Allowed AND L_Feedback.Feedback_Available AND NOT L_Convergence.Runtime_Converged;

    IF L_Diagnostics.Travel_Active THEN
        L_Diagnostics.Travel_Time_MS := 100;
    ELSE
        L_Diagnostics.Travel_Time_MS := 0;
    END_IF;

    IF L_Diagnostics.Travel_Time_MS > 4000 THEN
        L_Diagnostics.Travel_Timeout := TRUE;
        L_Diagnostics.Stuck_Suspected := TRUE;
    END_IF;

    IF L_Diagnostics.Travel_Timeout THEN
        L_Diagnostics.Diagnostics_Degraded := TRUE;
        L_Diagnostics.Escalation_Required := TRUE;
        L_Diagnostics.Failure_Count := 1;
        L_Diagnostics.Status_Code := 2;
        L_Diagnostics.Status_Text := 'Actuator travel timeout detected';
    ELSE
        L_Diagnostics.Status_Code := 0;
        L_Diagnostics.Status_Text := 'Actuator diagnostics healthy';
    END_IF;

    GVL_Water_Physical_Runtime.G_Convergence_State[L_i] := L_Convergence;
    GVL_Water_Physical_Runtime.G_Actuator_Diagnostics[L_i] := L_Diagnostics;

    L_Any_Convergence_Degraded := L_Any_Convergence_Degraded OR L_Convergence.Convergence_Degraded;
    L_Any_Diagnostics_Degraded := L_Any_Diagnostics_Degraded OR L_Diagnostics.Diagnostics_Degraded;
    L_Any_Escalation := L_Any_Escalation OR L_Convergence.Escalation_Required OR L_Diagnostics.Escalation_Required;
END_FOR;

GVL_Water_Physical_Runtime.G_Any_Convergence_Degraded := L_Any_Convergence_Degraded;
GVL_Water_Physical_Runtime.G_Any_Diagnostics_Degraded := L_Any_Diagnostics_Degraded;
GVL_Water_Physical_Runtime.G_Any_Escalation_Required := L_Any_Escalation;
GVL_Water_Physical_Runtime.G_Runtime_Valid := TRUE;
GVL_Water_Physical_Runtime.G_Last_Update_MS := VI_System_Time_MS;

IF L_Any_Escalation THEN
    GVL_Water_Physical_Runtime.G_Status_Code := 2;
    GVL_Water_Physical_Runtime.G_Status_Text := 'Physical runtime escalation active';
ELSIF L_Any_Convergence_Degraded THEN
    GVL_Water_Physical_Runtime.G_Status_Code := 1;
    GVL_Water_Physical_Runtime.G_Status_Text := 'Physical convergence degraded';
ELSE
    GVL_Water_Physical_Runtime.G_Status_Code := 0;
    GVL_Water_Physical_Runtime.G_Status_Text := 'Physical runtime healthy';
END_IF;
          
END_FUNCTION_BLOCK

FUNCTION_BLOCK FB_Heating_Policy_Priority_Bridge
  VAR_INPUT
    VI_Enable : BOOL;
    VI_Zone_Valves : ARRAY[1..GVL_CONSTANTS.C_MAX_HEATING_CIRCUITS] OF BOOL;
    VI_Zone_Configs : ARRAY[1..GVL_CONSTANTS.C_MAX_HEATING_CIRCUITS] OF ST_FloorHeating_Circuit_Config;
    VI_Manifold_Base_Priority : ARRAY[1..GVL_CONSTANTS.C_MAX_MANIFOLDS] OF INT;
    VI_Zone_Priority_Bias : ARRAY[1..GVL_CONSTANTS.C_MAX_ZONES] OF REAL;
    VI_Policy_Priority_Multiplier : REAL;
  END_VAR
  VAR_OUTPUT
    VO_Manifold_Effective_Priority : ARRAY[1..GVL_CONSTANTS.C_MAX_MANIFOLDS] OF INT;
    VO_Manifold_Priority_Bias_Applied : ARRAY[1..GVL_CONSTANTS.C_MAX_MANIFOLDS] OF REAL;
    VO_Bridge_Active : BOOL;
  END_VAR
  VAR
    L_i : INT;
    L_Manifold_ID : INT;
    L_Zone_ID : INT;
    L_Multiplier : REAL;
    L_Bias : REAL;
    L_Score : REAL;
    L_MaxScore : ARRAY[1..GVL_CONSTANTS.C_MAX_MANIFOLDS] OF REAL;
    L_HasActiveCircuit : ARRAY[1..GVL_CONSTANTS.C_MAX_MANIFOLDS] OF BOOL;
  END_VAR

            // ==============================================================================
// Heating policy priority bridge
//
// Bounded mapper from advisory zone policy to manifold allocation priority.
//
// IMPORTANT:
// - does NOT own demand;
// - does NOT create demand;
// - does NOT control pumps/valves;
// - does NOT write outputs;
// - does NOT bypass safety or service gates.
//
// Responsibility:
// - map circuit->zone policy bias into manifold effective priority;
// - keep the result bounded and deterministic;
// - provide a safe input for FB_Heating_Allocation_Filter.
// ==============================================================================



// Default passthrough state.
VO_Bridge_Active := FALSE;

FOR L_i := 1 TO GVL_CONSTANTS.C_MAX_MANIFOLDS DO
    VO_Manifold_Effective_Priority[L_i] := VI_Manifold_Base_Priority[L_i];
    VO_Manifold_Priority_Bias_Applied[L_i] := REAL#1.0;
    L_MaxScore[L_i] := REAL#0.0;
    L_HasActiveCircuit[L_i] := FALSE;
END_FOR;

IF NOT VI_Enable THEN
    RETURN;
END_IF;

L_Multiplier := VI_Policy_Priority_Multiplier;
IF L_Multiplier <= REAL#0.0 THEN
    L_Multiplier := REAL#1.0;
ELSIF L_Multiplier < REAL#0.3 THEN
    L_Multiplier := REAL#0.3;
ELSIF L_Multiplier > REAL#1.0 THEN
    L_Multiplier := REAL#1.0;
END_IF;

IF ABS(L_Multiplier - REAL#1.0) > REAL#0.001 THEN
    VO_Bridge_Active := TRUE;
END_IF;

FOR L_i := 1 TO GVL_CONSTANTS.C_MAX_HEATING_CIRCUITS DO
    IF VI_Zone_Valves[L_i] THEN
        L_Manifold_ID := TO_INT(VI_Zone_Configs[L_i].manifold_id);
        L_Zone_ID := TO_INT(VI_Zone_Configs[L_i].zone);

        IF (L_Manifold_ID >= 1)
           AND (L_Manifold_ID <= GVL_CONSTANTS.C_MAX_MANIFOLDS)
           AND (L_Zone_ID >= 1)
           AND (L_Zone_ID <= GVL_CONSTANTS.C_MAX_ZONES) THEN

            L_Bias := VI_Zone_Priority_Bias[L_Zone_ID];
            IF L_Bias <= REAL#0.0 THEN
                // Uninitialized advisory bias is treated as neutral.
                L_Bias := REAL#1.0;
            ELSIF L_Bias < REAL#0.3 THEN
                L_Bias := REAL#0.3;
            ELSIF L_Bias > REAL#1.5 THEN
                L_Bias := REAL#1.5;
            END_IF;

            IF ABS(L_Bias - REAL#1.0) > REAL#0.001 THEN
                VO_Bridge_Active := TRUE;
            END_IF;

            IF L_Bias > VO_Manifold_Priority_Bias_Applied[L_Manifold_ID] THEN
                VO_Manifold_Priority_Bias_Applied[L_Manifold_ID] := L_Bias;
            END_IF;

            L_Score := TO_REAL(VI_Manifold_Base_Priority[L_Manifold_ID]) * L_Multiplier * L_Bias;

            IF L_Score > L_MaxScore[L_Manifold_ID] THEN
                L_MaxScore[L_Manifold_ID] := L_Score;
            END_IF;

            L_HasActiveCircuit[L_Manifold_ID] := TRUE;
        END_IF;
    END_IF;
END_FOR;

FOR L_i := 1 TO GVL_CONSTANTS.C_MAX_MANIFOLDS DO
    IF L_HasActiveCircuit[L_i] THEN
        IF L_MaxScore[L_i] >= REAL#3.5 THEN
            VO_Manifold_Effective_Priority[L_i] := 4;
        ELSIF L_MaxScore[L_i] >= REAL#2.5 THEN
            VO_Manifold_Effective_Priority[L_i] := 3;
        ELSIF L_MaxScore[L_i] >= REAL#1.5 THEN
            VO_Manifold_Effective_Priority[L_i] := 2;
        ELSIF L_MaxScore[L_i] >= REAL#0.5 THEN
            VO_Manifold_Effective_Priority[L_i] := 1;
        ELSE
            VO_Manifold_Effective_Priority[L_i] := 0;
        END_IF;
    ELSE
        VO_Manifold_Effective_Priority[L_i] := VI_Manifold_Base_Priority[L_i];
        VO_Manifold_Priority_Bias_Applied[L_i] := REAL#1.0;
    END_IF;
END_FOR;

// >>> BULK_SYNC_ANCHOR: FB_Heating_Policy_Priority_Bridge <<<
          
END_FUNCTION_BLOCK

FUNCTION_BLOCK FB_Runtime_Node_Discovery
  VAR_INPUT
    VI_Enable : BOOL;
    VI_System_Time_MS : UDINT;
  END_VAR
  VAR
    L_i : INT;
    L_State : ST_Runtime_Node_Discovery_State;
    L_Any_Quarantine : BOOL;
    L_Any_Rejected : BOOL;
    L_Finalized_Runtime_Continuity : BOOL;
  END_VAR

            IF NOT VI_Enable THEN
    GVL_Runtime_Discovery.G_Runtime_Valid := FALSE;
    RETURN;
END_IF;

// Finalized runtime continuity proof chain.
L_Finalized_Runtime_Continuity :=
    GVL_SEMANTIC_PROGRESS.Semantic_Forward_Progress_Valid
    AND GVL_SEMANTIC_PROGRESS.Semantic_Execution_Continuity_OK
    AND NOT GVL_SEMANTIC_PROGRESS.Semantic_Progress_Lease_Expired
    AND NOT GVL_SEMANTIC_PROGRESS.Semantic_Progress_Quarantine_Active
    AND GVL_RUNTIME_SNAPSHOT.Snapshot_Frozen
    AND GVL_RUNTIME_SNAPSHOT.Snapshot_Publication_Allowed
    AND GVL_RUNTIME_SNAPSHOT.Snapshot_Copy_Valid
    AND GVL_RUNTIME_SNAPSHOT.Snapshot_Isolation_Valid
    AND NOT GVL_RUNTIME_SNAPSHOT.Snapshot_Mutation_Detected
    AND GVL_DISTRIBUTED_SNAPSHOT.Distributed_Publication_Reconciled
    AND GVL_DISTRIBUTED_SNAPSHOT.Distributed_Publication_Freeze_Valid
    AND GVL_DISTRIBUTED_SNAPSHOT.Distributed_Snapshot_Consistent
    AND GVL_DISTRIBUTED_COMMIT.Distributed_Commit_Valid
    AND GVL_DISTRIBUTED_COMMIT.Publication_Prepare_Valid
    AND GVL_DISTRIBUTED_COMMIT.Publication_Commit_Confirmed
    AND NOT GVL_DISTRIBUTED_COMMIT.Peer_Commit_Mismatch
    AND NOT GVL_DISTRIBUTED_COMMIT.Commit_Lease_Expired
    AND GVL_OUTPUT_EPOCH.Output_Publication_Valid
    AND GVL_OUTPUT_EPOCH.Output_Runtime_Epoch_Valid
    AND NOT GVL_OUTPUT_EPOCH.Output_Lease_Expired
    AND NOT GVL_OUTPUT_EPOCH.Output_Forced_Safe_Decay
    AND GVL_COMMAND_VERIFY.PreOutput_Barrier_OK
    AND NOT GVL_COMMAND_VERIFY.PreOutput_Block_IO;

FOR L_i := 1 TO 32 DO

    L_State := GVL_Runtime_Discovery.G_Discovery_State[L_i];

    IF L_State.Discovery_Active THEN

        L_State.Runtime_Valid := TRUE;
        L_State.Runtime_System_Time_MS := VI_System_Time_MS;

        L_State.Node_Discovered := TRUE;

        IF GVL_Distributed_Authority.G_Distributed_Safety_Barrier_OK
           AND NOT GVL_Runtime_Sessions.G_Any_Stale_Session
           AND L_Finalized_Runtime_Continuity THEN

            L_State.Node_Validated := TRUE;
            L_State.Node_Authorized := TRUE;

            L_State.Capability_Validated := TRUE;
            L_State.Execution_Domain_Assigned := TRUE;
            L_State.Deployment_Assigned := TRUE;

            L_State.Status_Code := 0;
            L_State.Status_Text :=
                'Runtime node discovery healthy';

        ELSE

            L_State.Node_Quarantined := TRUE;
            L_State.Discovery_Rejected := TRUE;

            L_Any_Quarantine := TRUE;
            L_Any_Rejected := TRUE;

            L_State.Status_Code := 2;
            L_State.Status_Text :=
                'Runtime node discovery rejected';

        END_IF;

        GVL_Runtime_Discovery.G_Discovery_State[L_i] :=
            L_State;

    END_IF;

END_FOR;

GVL_Runtime_Discovery.G_Any_Node_Quarantined :=
    L_Any_Quarantine;

GVL_Runtime_Discovery.G_Any_Discovery_Rejected :=
    L_Any_Rejected;

GVL_Runtime_Discovery.G_Runtime_Valid := TRUE;
GVL_Runtime_Discovery.G_Last_Update_MS := VI_System_Time_MS;

IF L_Any_Rejected THEN
    GVL_Runtime_Discovery.G_Status_Code := 2;
    GVL_Runtime_Discovery.G_Status_Text :=
        'Runtime discovery rejection detected';
ELSIF L_Any_Quarantine THEN
    GVL_Runtime_Discovery.G_Status_Code := 1;
    GVL_Runtime_Discovery.G_Status_Text :=
        'Runtime discovery quarantine active';
ELSE
    GVL_Runtime_Discovery.G_Status_Code := 0;
    GVL_Runtime_Discovery.G_Status_Text :=
        'Runtime discovery governance healthy';
END_IF;
          
END_FUNCTION_BLOCK

FUNCTION_BLOCK FB_Modbus_RTU_TX_Builder
  VAR_INPUT
    VI_Request_Valid : BOOL;
    VI_Slave_ID : BYTE;
    VI_Function_Code : E_Modbus_Function;
    VI_Start_Register : UINT;
    VI_Register_Count : UINT;
    VI_Write_Value : ARRAY[1..32] OF WORD;
  END_VAR
  VAR_OUTPUT
    VO_Frame : ST_Modbus_RTU_Frame;
    VO_Error : BOOL;
    VO_Error_Code : WORD;
  END_VAR
  VAR
    L_i : INT;
    L_j : INT;
    L_Pos : UINT;
    L_CRC : WORD;
    L_Byte_Count : UINT;
    L_Function_Byte : BYTE;
  END_VAR

            // ======================================================
// MODBUS RTU TX FRAME BUILDER
// ======================================================
// Builds Modbus RTU request frames only.
// This FB does not send data and does not modify response state.
// ======================================================

VO_Error := FALSE;
VO_Error_Code := 0;
VO_Frame.Valid := FALSE;
VO_Frame.Length := 0;
VO_Frame.CRC := 0;
L_Function_Byte := 0;

FOR L_i := 0 TO 255 DO
    VO_Frame.Data[L_i] := 0;
END_FOR;

IF NOT VI_Request_Valid THEN
    RETURN;
END_IF;

IF VI_Slave_ID = 0 THEN
    VO_Error := TRUE;
    VO_Error_Code := 16#0101;
    RETURN;
END_IF;

IF (VI_Register_Count = 0) OR (VI_Register_Count > 32) THEN
    VO_Error := TRUE;
    VO_Error_Code := 16#0102;
    RETURN;
END_IF;

CASE VI_Function_Code OF
    MB_FC03_READ_HOLDING_REGISTERS:
        L_Function_Byte := 3;
    MB_FC04_READ_INPUT_REGISTERS:
        L_Function_Byte := 4;
    MB_FC06_WRITE_SINGLE_REGISTER:
        L_Function_Byte := 6;
    MB_FC16_WRITE_MULTIPLE_REGISTERS:
        L_Function_Byte := 16;
ELSE
    VO_Error := TRUE;
    VO_Error_Code := 16#0104;
    RETURN;
END_CASE;

VO_Frame.Data[0] := VI_Slave_ID;
VO_Frame.Data[1] := L_Function_Byte;
VO_Frame.Data[2] := WORD_TO_BYTE(SHR(UINT_TO_WORD(VI_Start_Register), 8));
VO_Frame.Data[3] := WORD_TO_BYTE(UINT_TO_WORD(VI_Start_Register) AND 16#00FF);

CASE VI_Function_Code OF

    MB_FC03_READ_HOLDING_REGISTERS,
    MB_FC04_READ_INPUT_REGISTERS:

        VO_Frame.Data[4] := WORD_TO_BYTE(SHR(UINT_TO_WORD(VI_Register_Count), 8));
        VO_Frame.Data[5] := WORD_TO_BYTE(UINT_TO_WORD(VI_Register_Count) AND 16#00FF);
        VO_Frame.Length := 6;

    MB_FC06_WRITE_SINGLE_REGISTER:

        VO_Frame.Data[4] := WORD_TO_BYTE(SHR(VI_Write_Value[1], 8));
        VO_Frame.Data[5] := WORD_TO_BYTE(VI_Write_Value[1] AND 16#00FF);
        VO_Frame.Length := 6;

    MB_FC16_WRITE_MULTIPLE_REGISTERS:

        L_Byte_Count := VI_Register_Count * 2;

        IF L_Byte_Count > 64 THEN
            VO_Error := TRUE;
            VO_Error_Code := 16#0103;
            RETURN;
        END_IF;

        VO_Frame.Data[4] := WORD_TO_BYTE(SHR(UINT_TO_WORD(VI_Register_Count), 8));
        VO_Frame.Data[5] := WORD_TO_BYTE(UINT_TO_WORD(VI_Register_Count) AND 16#00FF);
        VO_Frame.Data[6] := UINT_TO_BYTE(L_Byte_Count);

        L_Pos := 7;

        FOR L_i := 1 TO UINT_TO_INT(VI_Register_Count) DO
            VO_Frame.Data[L_Pos] := WORD_TO_BYTE(SHR(VI_Write_Value[L_i], 8));
            VO_Frame.Data[L_Pos + 1] := WORD_TO_BYTE(VI_Write_Value[L_i] AND 16#00FF);
            L_Pos := L_Pos + 2;
        END_FOR;

        VO_Frame.Length := 7 + L_Byte_Count;

ELSE
    VO_Error := TRUE;
    VO_Error_Code := 16#0104;
    RETURN;
END_CASE;

// ======================================================
// INLINE MODBUS RTU CRC16
// ======================================================
L_CRC := 16#FFFF;

FOR L_i := 0 TO (UINT_TO_INT(VO_Frame.Length) - 1) DO

    L_CRC := L_CRC XOR BYTE_TO_WORD(VO_Frame.Data[L_i]);

    FOR L_j := 0 TO 7 DO
        IF (L_CRC AND 16#0001) <> 0 THEN
            L_CRC := SHR(L_CRC, 1);
            L_CRC := L_CRC XOR 16#A001;
        ELSE
            L_CRC := SHR(L_CRC, 1);
        END_IF;
    END_FOR;

END_FOR;

VO_Frame.CRC := L_CRC;
VO_Frame.Data[VO_Frame.Length] := WORD_TO_BYTE(L_CRC AND 16#00FF);
VO_Frame.Data[VO_Frame.Length + 1] := WORD_TO_BYTE(SHR(L_CRC, 8));
VO_Frame.Length := VO_Frame.Length + 2;
VO_Frame.Valid := TRUE;
          
END_FUNCTION_BLOCK

FUNCTION_BLOCK FB_MQTT_Runtime_Adapter
  VAR_INPUT
    VI_Enable : BOOL;
    VI_System_Time_MS : UDINT;
  END_VAR
  VAR
    L_Frame : ST_Runtime_Bus_Frame;
    L_TX_Index : UINT;
  END_VAR

            IF NOT VI_Enable THEN
    RETURN;
END_IF;

L_TX_Index := UDINT_TO_UINT(GVL_Runtime_Bus.G_Last_Sequence_Id);

IF (L_TX_Index >= 1)
   AND (L_TX_Index <= 128) THEN

    L_Frame := GVL_Runtime_Bus.G_TX_Frames[L_TX_Index];

    IF L_Frame.Frame_Valid THEN

        IF GVL_Distributed_Authority.G_Distributed_Safety_Barrier_OK
           AND NOT GVL_Runtime_Sessions.G_Any_Stale_Session THEN

            L_Frame.Frame_Ack_Received := TRUE;
            L_Frame.Replication_Consistent := TRUE;
            L_Frame.Status_Code := 0;

        ELSE

            L_Frame.Replication_Rejected := TRUE;
            L_Frame.Status_Code := 2;

        END_IF;

        GVL_Runtime_Bus.G_TX_Frames[L_TX_Index] := L_Frame;

    END_IF;

END_IF;
          
END_FUNCTION_BLOCK

FUNCTION_BLOCK FB_Runtime_Session_Governance
  VAR_INPUT
    VI_Enable : BOOL;
    VI_System_Time_MS : UDINT;
  END_VAR
  VAR
    L_i : INT;
    L_Session : ST_Runtime_Node_Session;
    L_Any_Stale : BOOL;
    L_Any_Quarantine : BOOL;
    L_Finalized_Runtime_Continuity : BOOL;
  END_VAR

            IF NOT VI_Enable THEN
    GVL_Runtime_Sessions.G_Runtime_Valid := FALSE;
    RETURN;
END_IF;

// Finalized runtime continuity proof chain.
L_Finalized_Runtime_Continuity :=
    GVL_SEMANTIC_PROGRESS.Semantic_Forward_Progress_Valid
    AND GVL_SEMANTIC_PROGRESS.Semantic_Execution_Continuity_OK
    AND NOT GVL_SEMANTIC_PROGRESS.Semantic_Progress_Lease_Expired
    AND NOT GVL_SEMANTIC_PROGRESS.Semantic_Progress_Quarantine_Active
    AND GVL_RUNTIME_SNAPSHOT.Snapshot_Frozen
    AND GVL_RUNTIME_SNAPSHOT.Snapshot_Publication_Allowed
    AND GVL_RUNTIME_SNAPSHOT.Snapshot_Copy_Valid
    AND GVL_RUNTIME_SNAPSHOT.Snapshot_Isolation_Valid
    AND NOT GVL_RUNTIME_SNAPSHOT.Snapshot_Mutation_Detected
    AND GVL_DISTRIBUTED_SNAPSHOT.Distributed_Publication_Reconciled
    AND GVL_DISTRIBUTED_SNAPSHOT.Distributed_Publication_Freeze_Valid
    AND GVL_DISTRIBUTED_SNAPSHOT.Distributed_Snapshot_Consistent
    AND GVL_DISTRIBUTED_COMMIT.Distributed_Commit_Valid
    AND GVL_DISTRIBUTED_COMMIT.Publication_Prepare_Valid
    AND GVL_DISTRIBUTED_COMMIT.Publication_Commit_Confirmed
    AND NOT GVL_DISTRIBUTED_COMMIT.Peer_Commit_Mismatch
    AND NOT GVL_DISTRIBUTED_COMMIT.Commit_Lease_Expired
    AND GVL_OUTPUT_EPOCH.Output_Publication_Valid
    AND GVL_OUTPUT_EPOCH.Output_Runtime_Epoch_Valid
    AND NOT GVL_OUTPUT_EPOCH.Output_Lease_Expired
    AND NOT GVL_OUTPUT_EPOCH.Output_Forced_Safe_Decay
    AND GVL_COMMAND_VERIFY.PreOutput_Barrier_OK
    AND NOT GVL_COMMAND_VERIFY.PreOutput_Block_IO;

GVL_Runtime_Sessions.G_Local_Session.Session_Valid := TRUE;
GVL_Runtime_Sessions.G_Local_Session.Session_Connected := TRUE;
GVL_Runtime_Sessions.G_Local_Session.Last_Heartbeat_MS :=
    VI_System_Time_MS;

GVL_Runtime_Sessions.G_Local_Session.Transport_Healthy :=
    GVL_Runtime_Bus.G_TX_Healthy
    AND L_Finalized_Runtime_Continuity;

GVL_Runtime_Sessions.G_Local_Session.Runtime_Replication_Healthy :=
    GVL_Distributed_Runtime.G_Distributed_Replication_Healthy
    AND L_Finalized_Runtime_Continuity;

GVL_Runtime_Sessions.G_Local_Session.Authority_Granted :=
    GVL_Distributed_Authority.G_Authority_State.Authority_Master_Elected
    AND L_Finalized_Runtime_Continuity;

FOR L_i := 1 TO 16 DO

    L_Session := GVL_Runtime_Sessions.G_Remote_Sessions[L_i];

    IF L_Session.Session_Valid THEN

        IF (VI_System_Time_MS - L_Session.Last_Heartbeat_MS) > 30000 THEN

            L_Session.Session_Stale := TRUE;
            L_Session.Session_Reconnect_Required := TRUE;

            L_Any_Stale := TRUE;

        END_IF;

        IF NOT L_Finalized_Runtime_Continuity THEN

            L_Session.Session_Stale := TRUE;
            L_Session.Session_Quarantined := TRUE;

            L_Any_Stale := TRUE;
            L_Any_Quarantine := TRUE;

        END_IF;

        IF L_Session.Session_Quarantined THEN
            L_Any_Quarantine := TRUE;
        END_IF;

        GVL_Runtime_Sessions.G_Remote_Sessions[L_i] :=
            L_Session;

    END_IF;

END_FOR;

GVL_Runtime_Sessions.G_Any_Stale_Session :=
    L_Any_Stale;

GVL_Runtime_Sessions.G_Any_Quarantined_Session :=
    L_Any_Quarantine;

GVL_Runtime_Sessions.G_Runtime_Valid := TRUE;
GVL_Runtime_Sessions.G_Last_Update_MS := VI_System_Time_MS;

IF L_Any_Quarantine THEN
    GVL_Runtime_Sessions.G_Status_Code := 2;
    GVL_Runtime_Sessions.G_Status_Text :=
        'Quarantined runtime session detected';
ELSIF L_Any_Stale THEN
    GVL_Runtime_Sessions.G_Status_Code := 1;
    GVL_Runtime_Sessions.G_Status_Text :=
        'Stale runtime session detected';
ELSE
    GVL_Runtime_Sessions.G_Status_Code := 0;
    GVL_Runtime_Sessions.G_Status_Text :=
        'Runtime session governance healthy';
END_IF;
          
END_FUNCTION_BLOCK

FUNCTION_BLOCK FB_Heating_Policy_Manager
  VAR_INPUT
    VI_System_Time_MS : UDINT;
    VI_System_Mode : E_System_Operating_Mode;
    VI_RootCause : E_Heating_RootCause;
    VI_RootConfidence : REAL;
    VI_Min_Hold_MS : UDINT;
    VI_Emergency_Stop : BOOL;
    VI_Gas_Safety : BOOL;
    VI_Room_Temp_Avg : REAL;
    VI_Floor_Temp_Avg : REAL;
    VI_Supply_Temp : REAL;
    VI_Return_Temp : REAL;
    VI_Target_Temp : REAL;
    VI_Room_Temps : ARRAY[1..GVL_CONSTANTS.C_MAX_ZONES] OF REAL;
    VI_Floor_Temps : ARRAY[1..GVL_CONSTANTS.C_MAX_ZONES] OF REAL;
  END_VAR
  VAR_OUTPUT
    VO_Policy_Mode : E_Heating_Policy_Mode;
    VO_Block_Heating : BOOL;
    VO_Target_Adjustment : REAL;
    VO_Priority_Multiplier : REAL;
    VO_Self_Tune_Active : BOOL;
    VO_Self_Tune_Level : INT;
    VO_Feedback_Stable : BOOL;
    VO_Feedback_Improving : BOOL;
    VO_Feedback_Quality : REAL;
  END_VAR
  VAR
    L_Raw_Mode : E_Heating_Policy_Mode;
    L_Raw_Block : BOOL;
    L_Raw_Target_Adjustment : REAL;
    L_Raw_Priority_Multiplier : REAL;
    L_Held_Mode : E_Heating_Policy_Mode;
    L_Held_Block : BOOL;
    L_Held_Target_Adjustment : REAL;
    L_Held_Priority_Multiplier : REAL;
    L_Last_Accept_MS : UDINT;
    L_Initialized : BOOL;
    L_Quality_Initialized : BOOL;
    L_Effective_Hold_MS : UDINT;
    L_Force_Immediate : BOOL;
    L_Same_Cause_Since : UDINT;
    L_Last_Cause : E_Heating_RootCause;
    L_Self_Level : INT;
    L_Room_Error : REAL;
    L_Supply_Error : REAL;
    L_DeltaT : REAL;
    L_Quality : REAL;
    L_Last_Quality : REAL;
    L_Improving : BOOL;
    L_Stable : BOOL;
    L_Last_Room_Avg : REAL;
    L_Trend : REAL;
    L_Filtered_Trend : REAL;
    L_Predictive_Adjustment : REAL;
    L_i : INT;
    L_Zone_Error : REAL;
    L_Zone_Quality : REAL;
    L_Zone_Desired_Level : INT;
    L_Zone_Last_Level_Accept_MS : ARRAY[1..GVL_CONSTANTS.C_MAX_ZONES] OF UDINT;
    L_Zone_Hold_MS : UDINT;
  END_VAR

            // ==============================================================================
// Ownership note
// ------------------------------------------------------------------------------
// This block owns only global policy mode/adjustment and policy quality/self-tune
// diagnostics. It does NOT own per-zone thermal fields, per-zone target adjustment,
// preheat request, or optimization demand values.
//
// Field owners:
// - FB_Heating_Thermal_Model: thermal response/demand/time/model confidence;
// - FB_Heating_Predictive_Controller: preheat-needed prediction;
// - FB_Heating_Optimizer: optimization scores/load diagnostics;
// - FB_Heating_Policy_Observer / FB_Heating_Schedule_Preheat: zone target policy;
// - FB_Heating_Policy_Manager: global policy and quality/self-level diagnostics.
// ==============================================================================

L_Zone_Hold_MS := VI_Min_Hold_MS / 2;
IF L_Zone_Hold_MS < 60000 THEN
    L_Zone_Hold_MS := 60000;
END_IF;

IF NOT L_Quality_Initialized THEN
    L_Last_Room_Avg := VI_Room_Temp_Avg;
    L_Filtered_Trend := 0.0;
    L_Same_Cause_Since := VI_System_Time_MS;
    L_Last_Cause := VI_RootCause;

    FOR L_i := 1 TO GVL_CONSTANTS.C_MAX_ZONES DO
        L_Zone_Last_Level_Accept_MS[L_i] := VI_System_Time_MS;
        GVL_HEATING_POLICY.G_Zone_Quality[L_i] := 0.0;
        GVL_HEATING_POLICY.G_Zone_Improving[L_i] := FALSE;
        GVL_HEATING_POLICY.G_Zone_Stable[L_i] := TRUE;
        GVL_HEATING_POLICY.G_Zone_Self_Level[L_i] := 0;
    END_FOR;

    L_Quality_Initialized := TRUE;
END_IF;

// ==============================================================================
// Global predictive adjustment based on aggregate room trend.
// ==============================================================================
L_Trend := VI_Room_Temp_Avg - L_Last_Room_Avg;
L_Last_Room_Avg := VI_Room_Temp_Avg;
L_Filtered_Trend := (L_Filtered_Trend * 0.8) + (L_Trend * 0.2);

L_Predictive_Adjustment := 0.0;
IF (L_Filtered_Trend < -0.03) AND (VI_Room_Temp_Avg < (VI_Target_Temp + 0.5)) THEN
    L_Predictive_Adjustment := 1.0;
ELSIF L_Filtered_Trend > 0.03 THEN
    L_Predictive_Adjustment := -0.5;
END_IF;

IF L_Predictive_Adjustment > 1.0 THEN
    L_Predictive_Adjustment := 1.0;
END_IF;
IF L_Predictive_Adjustment < -1.0 THEN
    L_Predictive_Adjustment := -1.0;
END_IF;

GVL_HEATING_POLICY.G_Policy_Predictive_Adjustment := L_Predictive_Adjustment;
GVL_HEATING_POLICY.G_Policy_Predictive_Active := ABS(L_Predictive_Adjustment) > 0.001;

// ==============================================================================
// Aggregate quality / feedback diagnostics.
// ==============================================================================
L_Room_Error := VI_Target_Temp - VI_Room_Temp_Avg;
L_Supply_Error := VI_Target_Temp - VI_Supply_Temp;
L_DeltaT := VI_Supply_Temp - VI_Return_Temp;
L_Quality := 0.0;

IF L_Room_Error > 1.0 THEN
    L_Quality := L_Quality + 2.0;
END_IF;
IF L_Supply_Error > 1.0 THEN
    L_Quality := L_Quality + 1.0;
END_IF;
IF L_DeltaT < 3.0 THEN
    L_Quality := L_Quality + 1.0;
END_IF;

L_Improving := L_Quality < L_Last_Quality;
L_Stable := L_Quality = 0.0;

// ==============================================================================
// Per-zone quality / self-level diagnostics only.
// Does not write target adjustment, thermal demand, time-to-heat, or preheat flags.
// ==============================================================================
FOR L_i := 1 TO GVL_CONSTANTS.C_MAX_ZONES DO
    L_Zone_Error := VI_Target_Temp - VI_Room_Temps[L_i];
    L_Zone_Quality := 0.0;

    IF L_Zone_Error > 1.0 THEN
        L_Zone_Quality := L_Zone_Quality + 2.0;
    END_IF;
    IF VI_Floor_Temps[L_i] < (VI_Target_Temp - 2.0) THEN
        L_Zone_Quality := L_Zone_Quality + 1.0;
    END_IF;

    GVL_HEATING_POLICY.G_Zone_Improving[L_i] :=
        L_Zone_Quality < GVL_HEATING_POLICY.G_Zone_Quality[L_i];

    GVL_HEATING_POLICY.G_Zone_Stable[L_i] :=
        L_Zone_Quality = 0.0;

    L_Zone_Desired_Level := GVL_HEATING_POLICY.G_Zone_Self_Level[L_i];

    IF GVL_HEATING_POLICY.G_Zone_Stable[L_i] THEN
        L_Zone_Desired_Level := 0;
    ELSIF GVL_HEATING_POLICY.G_Zone_Improving[L_i] THEN
        L_Zone_Desired_Level := GVL_HEATING_POLICY.G_Zone_Self_Level[L_i] - 1;
    ELSIF L_Zone_Quality >= 3.0 THEN
        L_Zone_Desired_Level := GVL_HEATING_POLICY.G_Zone_Self_Level[L_i] + 1;
    END_IF;

    IF L_Zone_Desired_Level > 2 THEN
        L_Zone_Desired_Level := 2;
    END_IF;
    IF L_Zone_Desired_Level < 0 THEN
        L_Zone_Desired_Level := 0;
    END_IF;

    IF L_Zone_Desired_Level <> GVL_HEATING_POLICY.G_Zone_Self_Level[L_i] THEN
        IF (VI_System_Time_MS - L_Zone_Last_Level_Accept_MS[L_i]) >= L_Zone_Hold_MS THEN
            GVL_HEATING_POLICY.G_Zone_Self_Level[L_i] := L_Zone_Desired_Level;
            L_Zone_Last_Level_Accept_MS[L_i] := VI_System_Time_MS;
        END_IF;
    END_IF;

    GVL_HEATING_POLICY.G_Zone_Quality[L_i] := L_Zone_Quality;
END_FOR;

// ==============================================================================
// Global self-level and policy mode.
// ==============================================================================
IF VI_RootCause <> L_Last_Cause THEN
    L_Same_Cause_Since := VI_System_Time_MS;
    L_Self_Level := 0;
END_IF;
L_Last_Cause := VI_RootCause;

IF L_Stable THEN
    L_Self_Level := 0;
ELSIF L_Improving THEN
    L_Self_Level := L_Self_Level - 1;
ELSIF (VI_System_Time_MS - L_Same_Cause_Since) > (VI_Min_Hold_MS * 2) AND (VI_RootConfidence > 0.8) AND (L_Quality >= 3.0) THEN
    L_Self_Level := L_Self_Level + 1;
END_IF;

IF L_Self_Level > 2 THEN
    L_Self_Level := 2;
END_IF;
IF L_Self_Level < 0 THEN
    L_Self_Level := 0;
END_IF;

L_Raw_Mode := E_Heating_Policy_Mode.HPM_NORMAL;
L_Raw_Block := FALSE;
L_Raw_Target_Adjustment := L_Predictive_Adjustment;
L_Raw_Priority_Multiplier := 1.0;
L_Force_Immediate := FALSE;

IF VI_Emergency_Stop OR VI_Gas_Safety THEN
    L_Raw_Mode := E_Heating_Policy_Mode.HPM_SAFETY_BLOCK;
    L_Raw_Block := TRUE;
    L_Raw_Target_Adjustment := 0.0;
    L_Raw_Priority_Multiplier := 1.0;
    L_Force_Immediate := TRUE;
ELSIF VI_RootCause = E_Heating_RootCause.RC_IO_OFFLINE THEN
    L_Raw_Mode := E_Heating_Policy_Mode.HPM_DEGRADED;
    L_Raw_Block := TRUE;
    L_Raw_Target_Adjustment := 0.0;
    L_Raw_Priority_Multiplier := 1.0;
    L_Force_Immediate := TRUE;
ELSIF VI_RootConfidence >= 0.6 THEN
    CASE VI_RootCause OF
        E_Heating_RootCause.RC_NO_HEAT_TRANSFER:
            L_Raw_Mode := E_Heating_Policy_Mode.HPM_DEGRADED;
            L_Raw_Target_Adjustment := L_Raw_Target_Adjustment + 3.0 + TO_REAL(L_Self_Level);
        E_Heating_RootCause.RC_PUMP_FAILURE:
            L_Raw_Mode := E_Heating_Policy_Mode.HPM_FAULT_ISOLATION;
            L_Raw_Priority_Multiplier := 0.5 - (0.1 * TO_REAL(L_Self_Level));
        E_Heating_RootCause.RC_VALVES_CLOSED:
            L_Raw_Mode := E_Heating_Policy_Mode.HPM_FAULT_ISOLATION;
            L_Raw_Target_Adjustment := L_Raw_Target_Adjustment - 2.0;
        E_Heating_RootCause.RC_NO_FLAME,
        E_Heating_RootCause.RC_BOILER_ERROR:
            L_Raw_Mode := E_Heating_Policy_Mode.HPM_DEGRADED;
            L_Raw_Priority_Multiplier := 0.7;
    ELSE
        IF VI_System_Mode = E_System_Operating_Mode.MODE_DEGRADED THEN
            L_Raw_Mode := E_Heating_Policy_Mode.HPM_DEGRADED;
        END_IF;
    END_CASE;
ELSE
    IF VI_System_Mode = E_System_Operating_Mode.MODE_DEGRADED THEN
        L_Raw_Mode := E_Heating_Policy_Mode.HPM_DEGRADED;
    END_IF;
END_IF;

IF L_Raw_Target_Adjustment > 5.0 THEN
    L_Raw_Target_Adjustment := 5.0;
END_IF;
IF L_Raw_Target_Adjustment < -3.0 THEN
    L_Raw_Target_Adjustment := -3.0;
END_IF;
IF L_Raw_Priority_Multiplier < 0.3 THEN
    L_Raw_Priority_Multiplier := 0.3;
END_IF;
IF L_Raw_Priority_Multiplier > 1.0 THEN
    L_Raw_Priority_Multiplier := 1.0;
END_IF;

L_Effective_Hold_MS := VI_Min_Hold_MS;
IF VI_RootConfidence >= 0.9 THEN
    L_Effective_Hold_MS := VI_Min_Hold_MS / 2;
END_IF;

IF NOT L_Initialized THEN
    L_Held_Mode := L_Raw_Mode;
    L_Held_Block := L_Raw_Block;
    L_Held_Target_Adjustment := L_Raw_Target_Adjustment;
    L_Held_Priority_Multiplier := L_Raw_Priority_Multiplier;
    L_Last_Accept_MS := VI_System_Time_MS;
    L_Initialized := TRUE;
ELSIF L_Force_Immediate THEN
    L_Held_Mode := L_Raw_Mode;
    L_Held_Block := L_Raw_Block;
    L_Held_Target_Adjustment := L_Raw_Target_Adjustment;
    L_Held_Priority_Multiplier := L_Raw_Priority_Multiplier;
    L_Last_Accept_MS := VI_System_Time_MS;
ELSIF (L_Raw_Mode <> L_Held_Mode) OR (ABS(L_Raw_Target_Adjustment - L_Held_Target_Adjustment) > 0.001) OR (ABS(L_Raw_Priority_Multiplier - L_Held_Priority_Multiplier) > 0.001) OR (L_Raw_Block <> L_Held_Block) THEN
    IF (VI_System_Time_MS - L_Last_Accept_MS) >= L_Effective_Hold_MS THEN
        L_Held_Mode := L_Raw_Mode;
        L_Held_Block := L_Raw_Block;
        L_Held_Target_Adjustment := L_Raw_Target_Adjustment;
        L_Held_Priority_Multiplier := L_Raw_Priority_Multiplier;
        L_Last_Accept_MS := VI_System_Time_MS;
    END_IF;
END_IF;

VO_Policy_Mode := L_Held_Mode;
VO_Block_Heating := L_Held_Block;
VO_Target_Adjustment := L_Held_Target_Adjustment;
VO_Priority_Multiplier := L_Held_Priority_Multiplier;
VO_Self_Tune_Active := L_Self_Level > 0;
VO_Self_Tune_Level := L_Self_Level;
VO_Feedback_Stable := L_Stable;
VO_Feedback_Improving := L_Improving;
VO_Feedback_Quality := L_Quality;

L_Last_Quality := L_Quality;
          
END_FUNCTION_BLOCK

FUNCTION_BLOCK FB_Cluster_Runtime_FSM
  VAR_INPUT
    VI_Enable : BOOL;
    VI_System_Time_MS : UDINT;
  END_VAR
  VAR
    L_Finalized_Runtime_Continuity : BOOL;
  END_VAR

            IF NOT VI_Enable THEN
    GVL_Cluster_Runtime_FSM.G_Runtime_Valid := FALSE;
    RETURN;
END_IF;

// Finalized runtime continuity proof chain.
L_Finalized_Runtime_Continuity :=
    GVL_SEMANTIC_PROGRESS.Semantic_Forward_Progress_Valid
    AND GVL_SEMANTIC_PROGRESS.Semantic_Execution_Continuity_OK
    AND NOT GVL_SEMANTIC_PROGRESS.Semantic_Progress_Lease_Expired
    AND NOT GVL_SEMANTIC_PROGRESS.Semantic_Progress_Quarantine_Active
    AND GVL_RUNTIME_SNAPSHOT.Snapshot_Frozen
    AND GVL_RUNTIME_SNAPSHOT.Snapshot_Publication_Allowed
    AND GVL_RUNTIME_SNAPSHOT.Snapshot_Copy_Valid
    AND GVL_RUNTIME_SNAPSHOT.Snapshot_Isolation_Valid
    AND NOT GVL_RUNTIME_SNAPSHOT.Snapshot_Mutation_Detected
    AND GVL_DISTRIBUTED_SNAPSHOT.Distributed_Publication_Reconciled
    AND GVL_DISTRIBUTED_SNAPSHOT.Distributed_Publication_Freeze_Valid
    AND GVL_DISTRIBUTED_SNAPSHOT.Distributed_Snapshot_Consistent
    AND GVL_DISTRIBUTED_COMMIT.Distributed_Commit_Valid
    AND GVL_DISTRIBUTED_COMMIT.Publication_Prepare_Valid
    AND GVL_DISTRIBUTED_COMMIT.Publication_Commit_Confirmed
    AND NOT GVL_DISTRIBUTED_COMMIT.Peer_Commit_Mismatch
    AND NOT GVL_DISTRIBUTED_COMMIT.Commit_Lease_Expired
    AND GVL_OUTPUT_EPOCH.Output_Publication_Valid
    AND GVL_OUTPUT_EPOCH.Output_Runtime_Epoch_Valid
    AND NOT GVL_OUTPUT_EPOCH.Output_Lease_Expired
    AND NOT GVL_OUTPUT_EPOCH.Output_Forced_Safe_Decay
    AND GVL_COMMAND_VERIFY.PreOutput_Barrier_OK
    AND NOT GVL_COMMAND_VERIFY.PreOutput_Block_IO;

// Reset runtime states.
GVL_Cluster_Runtime_FSM.G_State_Startup := FALSE;
GVL_Cluster_Runtime_FSM.G_State_Discovery := FALSE;
GVL_Cluster_Runtime_FSM.G_State_Synchronization := FALSE;
GVL_Cluster_Runtime_FSM.G_State_Operational := FALSE;
GVL_Cluster_Runtime_FSM.G_State_Degraded := FALSE;
GVL_Cluster_Runtime_FSM.G_State_Observer_Only := FALSE;
GVL_Cluster_Runtime_FSM.G_State_Recovery_Lock := FALSE;
GVL_Cluster_Runtime_FSM.G_State_Quarantine := FALSE;

// Startup state.
IF NOT GVL_Distributed_Runtime.G_Runtime_Valid THEN

    GVL_Cluster_Runtime_FSM.G_State_Startup := TRUE;

    GVL_Cluster_Runtime_FSM.G_Status_Code := 1;
    GVL_Cluster_Runtime_FSM.G_Status_Text :=
        'Cluster runtime startup';

ELSIF GVL_Runtime_Discovery.G_Runtime_Valid
   AND NOT GVL_Runtime_Discovery.G_Any_Discovery_Rejected THEN

    GVL_Cluster_Runtime_FSM.G_State_Discovery := TRUE;

    GVL_Cluster_Runtime_FSM.G_Status_Code := 2;
    GVL_Cluster_Runtime_FSM.G_Status_Text :=
        'Cluster runtime discovery';

END_IF;

// Synchronization state.
IF GVL_Runtime_Bus.G_TX_Healthy
   AND GVL_Runtime_Bus.G_RX_Healthy THEN

    GVL_Cluster_Runtime_FSM.G_State_Synchronization := TRUE;

END_IF;

// Operational state.
IF GVL_Distributed_Execution_Gates.G_Can_Execute
   AND GVL_Distributed_Execution_Gates.G_Can_Orchestrate
   AND L_Finalized_Runtime_Continuity THEN

    GVL_Cluster_Runtime_FSM.G_State_Operational := TRUE;

    GVL_Cluster_Runtime_FSM.G_Status_Code := 0;
    GVL_Cluster_Runtime_FSM.G_Status_Text :=
        'Cluster runtime operational';

END_IF;

// Degraded state.
IF GVL_Cluster_Safety_Barrier.G_Cluster_Execution_Blocked THEN

    GVL_Cluster_Runtime_FSM.G_State_Degraded := TRUE;

    GVL_Cluster_Runtime_FSM.G_Status_Code := 10;
    GVL_Cluster_Runtime_FSM.G_Status_Text :=
        'Cluster runtime degraded';

END_IF;

// Observer-only state.
IF GVL_Distributed_Authority.G_Authority_State.Authority_Observer_Only THEN

    GVL_Cluster_Runtime_FSM.G_State_Observer_Only := TRUE;

    GVL_Cluster_Runtime_FSM.G_Status_Code := 11;
    GVL_Cluster_Runtime_FSM.G_Status_Text :=
        'Cluster runtime observer-only';

END_IF;

// Recovery lock state.
IF GVL_Distributed_Recovery_Lock.G_Recovery_Execution_Blocked THEN

    GVL_Cluster_Runtime_FSM.G_State_Recovery_Lock := TRUE;

    GVL_Cluster_Runtime_FSM.G_Status_Code := 12;
    GVL_Cluster_Runtime_FSM.G_Status_Text :=
        'Cluster runtime recovery-locked';

END_IF;

// Quarantine state.
IF GVL_Runtime_Discovery.G_Any_Node_Quarantined THEN

    GVL_Cluster_Runtime_FSM.G_State_Quarantine := TRUE;

    GVL_Cluster_Runtime_FSM.G_Status_Code := 13;
    GVL_Cluster_Runtime_FSM.G_Status_Text :=
        'Cluster runtime quarantined';

END_IF;

GVL_Cluster_Runtime_FSM.G_Runtime_Valid := TRUE;
GVL_Cluster_Runtime_FSM.G_Last_Update_MS := VI_System_Time_MS;
          
END_FUNCTION_BLOCK

FUNCTION_BLOCK FB_SHA1
  VAR_INPUT
    Length : INT;
  END_VAR
  VAR_OUTPUT
    Hash : ARRAY[0..19] OF BYTE;
  END_VAR
  VAR_IN_OUT
    Data : ARRAY[0..127] OF BYTE;
  END_VAR
  VAR
    H0, H1, H2, H3, H4 : DWORD;
    A, B, C, D, E, F, K, Temp : DWORD;
    W : ARRAY[0..79] OF DWORD;
    i, j, t : INT;
    PaddedData : ARRAY[0..127] OF BYTE;
    PaddedLength : INT;
    NumBlocks : INT;
    BlockOffset : INT;
  END_VAR

            // Initialize variables
H0 := 16#67452301;
H1 := 16#EFCDAB89;
H2 := 16#98BADCFE;
H3 := 16#10325476;
H4 := 16#C3D2E1F0;

// Pre-processing
FOR i := 0 TO Length - 1 DO
    PaddedData[i] := Data[i];
END_FOR;

// Append the bit '1' to the message
PaddedData[Length] := 16#80;

// Append 0 <= k < 512 bits '0', such that the resulting message length in bits
// is congruent to -64 ≡ 448 (mod 512)
PaddedLength := Length + 1;
WHILE (PaddedLength MOD 64) <> 56 DO
    PaddedData[PaddedLength] := 0;
    PaddedLength := PaddedLength + 1;
END_WHILE;

// Append length of message (before pre-processing), in bits, as 64-bit big-endian integer
// Since our message is small (max 127 bytes), we only need the lower 32 bits
Temp := TO_DWORD(Length * 8);
PaddedData[PaddedLength] := 0;
PaddedData[PaddedLength+1] := 0;
PaddedData[PaddedLength+2] := 0;
PaddedData[PaddedLength+3] := 0;
PaddedData[PaddedLength+4] := TO_BYTE(SHR(Temp, 24));
PaddedData[PaddedLength+5] := TO_BYTE(SHR(Temp, 16));
PaddedData[PaddedLength+6] := TO_BYTE(SHR(Temp, 8));
PaddedData[PaddedLength+7] := TO_BYTE(Temp);
PaddedLength := PaddedLength + 8;

NumBlocks := PaddedLength / 64;

// Process the message in successive 512-bit chunks
FOR i := 0 TO NumBlocks - 1 DO
    BlockOffset := i * 64;
    
    // Break chunk into sixteen 32-bit big-endian words w[i], 0 <= i <= 15
    FOR j := 0 TO 15 DO
        W[j] := SHL(TO_DWORD(PaddedData[BlockOffset + j*4]), 24) OR
                SHL(TO_DWORD(PaddedData[BlockOffset + j*4 + 1]), 16) OR
                SHL(TO_DWORD(PaddedData[BlockOffset + j*4 + 2]), 8) OR
                TO_DWORD(PaddedData[BlockOffset + j*4 + 3]);
    END_FOR;
    
    // Message schedule: extend the sixteen 32-bit words into eighty 32-bit words
    FOR j := 16 TO 79 DO
        Temp := W[j-3] XOR W[j-8] XOR W[j-14] XOR W[j-16];
        W[j] := SHL(Temp, 1) OR SHR(Temp, 31); // Left rotate by 1
    END_FOR;
    
    // Initialize hash value for this chunk
    A := H0;
    B := H1;
    C := H2;
    D := H3;
    E := H4;
    
    // Main loop
    FOR j := 0 TO 79 DO
        IF j <= 19 THEN
            F := (B AND C) OR ((NOT B) AND D);
            K := 16#5A827999;
        ELSIF j <= 39 THEN
            F := B XOR C XOR D;
            K := 16#6ED9EBA1;
        ELSIF j <= 59 THEN
            F := (B AND C) OR (B AND D) OR (C AND D);
            K := 16#8F1BBCDC;
        ELSE
            F := B XOR C XOR D;
            K := 16#CA62C1D6;
        END_IF;
        
        Temp := (SHL(A, 5) OR SHR(A, 27)) + F + E + K + W[j];
        E := D;
        D := C;
        C := SHL(B, 30) OR SHR(B, 2);
        B := A;
        A := Temp;
    END_FOR;
    
    // Add this chunk's hash to result so far
    H0 := H0 + A;
    H1 := H1 + B;
    H2 := H2 + C;
    H3 := H3 + D;
    H4 := H4 + E;
END_FOR;

// Produce the final hash value (big-endian)
Hash[0] := TO_BYTE(SHR(H0, 24)); Hash[1] := TO_BYTE(SHR(H0, 16)); Hash[2] := TO_BYTE(SHR(H0, 8)); Hash[3] := TO_BYTE(H0);
Hash[4] := TO_BYTE(SHR(H1, 24)); Hash[5] := TO_BYTE(SHR(H1, 16)); Hash[6] := TO_BYTE(SHR(H1, 8)); Hash[7] := TO_BYTE(H1);
Hash[8] := TO_BYTE(SHR(H2, 24)); Hash[9] := TO_BYTE(SHR(H2, 16)); Hash[10] := TO_BYTE(SHR(H2, 8)); Hash[11] := TO_BYTE(H2);
Hash[12] := TO_BYTE(SHR(H3, 24)); Hash[13] := TO_BYTE(SHR(H3, 16)); Hash[14] := TO_BYTE(SHR(H3, 8)); Hash[15] := TO_BYTE(H3);
Hash[16] := TO_BYTE(SHR(H4, 24)); Hash[17] := TO_BYTE(SHR(H4, 16)); Hash[18] := TO_BYTE(SHR(H4, 8)); Hash[19] := TO_BYTE(H4);
          
END_FUNCTION_BLOCK

FUNCTION_BLOCK FB_Heating_Safety_Gate
  VAR_INPUT
    VI_System_Mode : E_System_Operating_Mode;
    VI_Emergency_Stop : BOOL;
    VI_Gas_Safety_Stop : BOOL;
    VI_IO_Failsafe_Active : BOOL;
    VI_Outdoor_Temp : REAL;
    VI_Freeze_Threshold : REAL;
  END_VAR
  VAR_OUTPUT
    VO_Block_Normal_Heating : BOOL;
    VO_Gas_Safety_Active : BOOL;
    VO_Emergency_Safe_Stop_Active : BOOL;
    VO_IO_Failsafe_Active : BOOL;
    VO_Freeze_Mode_Active : BOOL;
    VO_Freeze_Target_Supply : REAL;
    VO_Outdoor_Temp_Valid : BOOL;
  END_VAR
  VAR_IN_OUT
    VI_Floor_Temps : ARRAY[1..GVL_CONSTANTS.C_MAX_HEATING_CIRCUITS] OF REAL;
  END_VAR
  VAR
    L_i : INT;
    L_Outdoor_Temp_Safe : REAL;
  END_VAR

            // ==============================================================================
// Heating safety gate helper
// ==============================================================================



VO_Gas_Safety_Active := VI_Gas_Safety_Stop;
VO_Emergency_Safe_Stop_Active := VI_Emergency_Stop OR (VI_System_Mode = E_System_Operating_Mode.MODE_SAFE_STOP);
VO_IO_Failsafe_Active := VI_IO_Failsafe_Active;

// REAL validity guard: NaN fails self-equality; extreme values are rejected as sensor faults.
VO_Outdoor_Temp_Valid := (VI_Outdoor_Temp = VI_Outdoor_Temp) AND (VI_Outdoor_Temp > -80.0) AND (VI_Outdoor_Temp < 80.0);
IF VO_Outdoor_Temp_Valid THEN
    L_Outdoor_Temp_Safe := VI_Outdoor_Temp;
ELSE
    L_Outdoor_Temp_Safe := 20.0;
    GVL_STATE.G_Heating_Sensor_Fault := TRUE;
END_IF;

VO_Block_Normal_Heating := VO_Gas_Safety_Active OR VO_Emergency_Safe_Stop_Active OR VO_IO_Failsafe_Active;
VO_Freeze_Mode_Active := (VI_System_Mode = E_System_Operating_Mode.MODE_FREEZE_PROTECTION) OR (L_Outdoor_Temp_Safe < -5.0);

FOR L_i := 1 TO GVL_CONSTANTS.C_MAX_HEATING_CIRCUITS DO
    IF VI_Floor_Temps[L_i] < 7.0 THEN
        VO_Freeze_Mode_Active := TRUE;
    END_IF;
END_FOR;

IF VO_Freeze_Mode_Active THEN
    VO_Freeze_Target_Supply := LIMIT(20.0, VI_Freeze_Threshold + 2.0, 35.0);
ELSE
    VO_Freeze_Target_Supply := 0.0;
END_IF;

// >>> BULK_SYNC_ANCHOR: FB_Heating_Safety_Gate <<<
          
END_FUNCTION_BLOCK

FUNCTION_BLOCK FB_Heating_Output_Projection
  VAR_INPUT
    VI_Zone_Valves : ARRAY[1..GVL_CONSTANTS.C_MAX_HEATING_CIRCUITS] OF BOOL;
    VI_Manifold_Pumps : ARRAY[1..GVL_CONSTANTS.C_MAX_MANIFOLDS] OF BOOL;
    VI_Manifold_Valves : ARRAY[1..GVL_CONSTANTS.C_MAX_MANIFOLDS] OF REAL;
    VI_DHW_Heating_Pump : BOOL;
    VI_DHW_Circ_Pump : BOOL;
    VI_Backup_Circulation_Pump : BOOL;
    VI_Electric_Heater_Enable : BOOL;
  END_VAR
  VAR
    L_i : INT;
  END_VAR

            FOR L_i := 1 TO GVL_CONSTANTS.C_MAX_HEATING_CIRCUITS DO
    GVL_HEATING_OUTPUT.DO_Zone_Valves[L_i] := VI_Zone_Valves[L_i];
END_FOR;

FOR L_i := 1 TO GVL_CONSTANTS.C_MAX_MANIFOLDS DO
    GVL_HEATING_OUTPUT.DO_Manifold_Pumps[L_i] := VI_Manifold_Pumps[L_i];
    GVL_HEATING_OUTPUT.AO_Manifold_Valves[L_i] := REAL_TO_UINT(VI_Manifold_Valves[L_i] * 1000.0);
END_FOR;

GVL_HEATING_OUTPUT.DO_DHW_Heating_Pump := VI_DHW_Heating_Pump;
GVL_HEATING_OUTPUT.DO_DHW_Circ_Pump := VI_DHW_Circ_Pump;
GVL_HEATING_OUTPUT.DO_Backup_Circulation_Pump := VI_Backup_Circulation_Pump;
GVL_HEATING_OUTPUT.DO_Electric_Heater_Enable := VI_Electric_Heater_Enable;

// >>> BULK_SYNC_ANCHOR: FB_Heating_Output_Projection <<<
          
END_FUNCTION_BLOCK

FUNCTION_BLOCK FB_Water_Isolation_Intent_Builder
  VAR_INPUT
    VI_Enable : BOOL;
  END_VAR
  VAR
    L_i : INT;
    L_State : ST_Water_Isolation_Runtime_State;
    L_Any_Selective : BOOL;
    L_Global_Fallback : BOOL;
  END_VAR

            IF NOT VI_Enable THEN
    GVL_Water_Isolation_Intent.G_Intent_Valid := FALSE;
    RETURN;
END_IF;

L_Any_Selective := FALSE;
L_Global_Fallback := FALSE;

FOR L_i := 1 TO GVL_CONSTANTS.C_MAX_FLOOD_SENSORS DO

    L_State := GVL_Water_Isolation_Runtime.G_Isolation_Runtime_State[L_i];

    GVL_Water_Isolation_Intent.G_Zone_Close_Requested[L_i] := FALSE;
    GVL_Water_Isolation_Intent.G_Valve_Group_Close_Requested[L_i] := FALSE;

    IF L_State.Selective_Isolation_Requested THEN

        IF (L_State.Hydraulic_Zone_Id >= 1)
           AND (L_State.Hydraulic_Zone_Id <= GVL_CONSTANTS.C_MAX_FLOOD_SENSORS) THEN

            GVL_Water_Isolation_Intent.G_Zone_Close_Requested[
                L_State.Hydraulic_Zone_Id
            ] := TRUE;

        END_IF;

        IF (L_State.Valve_Group_Id >= 1)
           AND (L_State.Valve_Group_Id <= GVL_CONSTANTS.C_MAX_FLOOD_SENSORS) THEN

            GVL_Water_Isolation_Intent.G_Valve_Group_Close_Requested[
                L_State.Valve_Group_Id
            ] := TRUE;

        END_IF;

        L_Any_Selective := TRUE;

    END_IF;

    IF L_State.Global_Isolation_Requested THEN
        L_Global_Fallback := TRUE;
    END_IF;

END_FOR;

GVL_Water_Isolation_Intent.G_Global_Isolation_Requested :=
    L_Global_Fallback;

GVL_Water_Isolation_Intent.G_Intent_Valid := TRUE;

IF L_Global_Fallback THEN
    GVL_Water_Isolation_Intent.G_Status_Code := 2;
    GVL_Water_Isolation_Intent.G_Status_Text :=
        'Global isolation fallback requested';
ELSIF L_Any_Selective THEN
    GVL_Water_Isolation_Intent.G_Status_Code := 1;
    GVL_Water_Isolation_Intent.G_Status_Text :=
        'Localized isolation intent available';
ELSE
    GVL_Water_Isolation_Intent.G_Status_Code := 0;
    GVL_Water_Isolation_Intent.G_Status_Text :=
        'No isolation intent active';
END_IF;
          
END_FUNCTION_BLOCK

FUNCTION_BLOCK FB_Distributed_Execution_Gates_Runtime
  VAR_INPUT
    VI_Enable : BOOL;
    VI_System_Time_MS : UDINT;
  END_VAR
  VAR
    L_Allow : BOOL;
    L_Observer_Only : BOOL;
    L_Semantic_Continuity_Valid : BOOL;
    L_Finalized_Publication_Continuity : BOOL;
  END_VAR

            IF NOT VI_Enable THEN
    GVL_Distributed_Execution_Gates.G_Runtime_Valid := FALSE;
    RETURN;
END_IF;

// Observer-only runtime semantics.
// Observer nodes may:
//   - observe runtime state;
//   - receive publications;
//   - participate in diagnostics.
//
// Observer nodes must NEVER:
//   - execute orchestration;
//   - own projections;
//   - execute recovery;
//   - publish physical outputs.
L_Observer_Only :=
    GVL_Distributed_Authority.G_Authority_State.Authority_Observer_Only;

// Semantic continuity authority.
L_Semantic_Continuity_Valid :=
    GVL_SEMANTIC_PROGRESS.Semantic_Forward_Progress_Valid
    AND GVL_SEMANTIC_PROGRESS.Semantic_Execution_Continuity_OK
    AND NOT GVL_SEMANTIC_PROGRESS.Semantic_Progress_Lease_Expired
    AND NOT GVL_SEMANTIC_PROGRESS.Semantic_Progress_Quarantine_Active
    AND NOT GVL_SEMANTIC_PROGRESS.Semantic_Replay_Suspected
    AND NOT GVL_SEMANTIC_PROGRESS.Semantic_Livelock_Suspected
    AND NOT GVL_SEMANTIC_PROGRESS.Semantic_Deadlock_Suspected;

// Finalized publication proof chain.
L_Finalized_Publication_Continuity :=
    GVL_RUNTIME_SNAPSHOT.Snapshot_Frozen
    AND GVL_RUNTIME_SNAPSHOT.Snapshot_Publication_Allowed
    AND GVL_RUNTIME_SNAPSHOT.Snapshot_Copy_Valid
    AND GVL_RUNTIME_SNAPSHOT.Snapshot_Isolation_Valid
    AND NOT GVL_RUNTIME_SNAPSHOT.Snapshot_Mutation_Detected
    AND GVL_DISTRIBUTED_SNAPSHOT.Distributed_Publication_Reconciled
    AND GVL_DISTRIBUTED_SNAPSHOT.Distributed_Publication_Freeze_Valid
    AND GVL_DISTRIBUTED_SNAPSHOT.Distributed_Snapshot_Consistent
    AND GVL_DISTRIBUTED_COMMIT.Distributed_Commit_Valid
    AND GVL_DISTRIBUTED_COMMIT.Publication_Prepare_Valid
    AND GVL_DISTRIBUTED_COMMIT.Publication_Commit_Confirmed
    AND NOT GVL_DISTRIBUTED_COMMIT.Peer_Commit_Mismatch
    AND NOT GVL_DISTRIBUTED_COMMIT.Commit_Lease_Expired
    AND GVL_OUTPUT_EPOCH.Output_Publication_Valid
    AND GVL_OUTPUT_EPOCH.Output_Runtime_Epoch_Valid
    AND NOT GVL_OUTPUT_EPOCH.Output_Lease_Expired
    AND NOT GVL_OUTPUT_EPOCH.Output_Forced_Safe_Decay
    AND GVL_COMMAND_VERIFY.PreOutput_Barrier_OK
    AND NOT GVL_COMMAND_VERIFY.PreOutput_Block_IO;

L_Allow :=
    NOT GVL_Cluster_Safety_Barrier.G_Cluster_Execution_Blocked
    AND GVL_Distributed_Authority.G_Authority_State.Authority_Master_Elected
    AND NOT GVL_Distributed_Runtime.G_Split_Brain_Suspected
    AND NOT GVL_Distributed_Projection_Ownership.G_Any_Ownership_Conflict
    AND NOT GVL_Runtime_Sessions.G_Any_Stale_Session
    AND L_Semantic_Continuity_Valid
    AND L_Finalized_Publication_Continuity
    AND NOT L_Observer_Only;

GVL_Distributed_Execution_Gates.G_Can_Replicate :=
    GVL_Runtime_Bus.G_TX_Healthy
    AND GVL_Runtime_Bus.G_RX_Healthy;

GVL_Distributed_Execution_Gates.G_Can_Execute :=
    L_Allow;

GVL_Distributed_Execution_Gates.G_Can_Orchestrate :=
    L_Allow
    AND GVL_Distributed_Orchestration.G_Distributed_Scheduler_Healthy;

GVL_Distributed_Execution_Gates.G_Can_Recover :=
    L_Allow
    AND NOT GVL_Distributed_Recovery_Lock.G_Recovery_Execution_Blocked;

GVL_Distributed_Execution_Gates.G_Can_Rollback :=
    L_Allow
    AND NOT GVL_Distributed_Recovery_Lock.G_Rollback_Execution_Blocked;

GVL_Distributed_Execution_Gates.G_Can_Own_Projection :=
    L_Allow
    AND NOT GVL_Distributed_Projection_Ownership.G_Any_Projection_Blocked;

GVL_Distributed_Execution_Gates.G_Runtime_Valid := TRUE;
GVL_Distributed_Execution_Gates.G_Last_Update_MS :=
    VI_System_Time_MS;

IF L_Observer_Only THEN

    GVL_Distributed_Execution_Gates.G_Status_Code := 2;
    GVL_Distributed_Execution_Gates.G_Status_Text :=
        'Distributed runtime observer-only';

ELSIF L_Allow THEN

    GVL_Distributed_Execution_Gates.G_Status_Code := 0;
    GVL_Distributed_Execution_Gates.G_Status_Text :=
        'Distributed execution gates open';

ELSE

    GVL_Distributed_Execution_Gates.G_Status_Code := 1;
    GVL_Distributed_Execution_Gates.G_Status_Text :=
        'Distributed execution gates restricted';

END_IF;
          
END_FUNCTION_BLOCK

FUNCTION_BLOCK FB_Water_Runtime_Hardening
  VAR_INPUT
    VI_Enable : BOOL;
    VI_System_Time_MS : UDINT;
  END_VAR
  VAR
    L_i : INT;
    L_FSM : ST_Water_Recovery_FSM_State;
    L_Event : ST_Water_Event_Log_Record;
    L_Any_Rollback : BOOL;
    L_Any_Escalation : BOOL;
  END_VAR

            IF NOT VI_Enable THEN
    GVL_Water_Runtime_Hardening.G_Runtime_Valid := FALSE;
    RETURN;
END_IF;

FOR L_i := 1 TO GVL_CONSTANTS.C_MAX_FLOOD_SENSORS DO

    // Recovery FSM.
    L_FSM := (Runtime_Valid := TRUE);

    L_FSM.Runtime_System_Time_MS :=
        VI_System_Time_MS;

    L_FSM.Recovery_Domain_Id :=
        GVL_Water_Topology_Config.G_Config_Record[L_i].Recovery_Domain_Id;

    L_FSM.Recovery_Requested :=
        GVL_INTENT_SAFETY.I_Water_Selective_Recovery_Allowed;

    L_FSM.Recovery_Sequencing_Active :=
        GVL_Water_Orchestration.G_Orchestration_State[L_i].Recovery_Sequence_Active;

    L_FSM.Recovery_Verification_Window_Active :=
        GVL_Water_Orchestration.G_Orchestration_State[L_i].Observation_Window_Active;

    // Conservative runtime hardening.
    IF GVL_Water_Physical_Runtime.G_Convergence_State[L_i].Escalation_Required THEN

        L_FSM.Rollback_Required := TRUE;
        L_FSM.Escalation_Required := TRUE;
        L_FSM.Operator_Ack_Required := TRUE;
        L_FSM.Recovery_Denied := TRUE;
        L_FSM.FSM_State := 100;

        L_FSM.Status_Code := 2;
        L_FSM.Status_Text :=
            'Recovery rollback escalation active';

    ELSIF L_FSM.Recovery_Requested THEN

        L_FSM.Recovery_Completed := TRUE;
        L_FSM.FSM_State := 10;

        L_FSM.Status_Code := 1;
        L_FSM.Status_Text :=
            'Recovery sequencing active';

    ELSE

        L_FSM.FSM_State := 0;

        L_FSM.Status_Code := 0;
        L_FSM.Status_Text :=
            'Recovery FSM idle';

    END_IF;

    GVL_Water_Runtime_Hardening.G_Recovery_FSM[L_i] :=
        L_FSM;

    // Runtime event publication.
    IF L_i <= 128 THEN

        L_Event := (Runtime_Valid := TRUE);

        L_Event.Event_Time_MS := VI_System_Time_MS;
        L_Event.Event_Id := TO_UINT(L_i);

        IF L_FSM.Escalation_Required THEN
            L_Event.Event_Text :=
                'Water runtime escalation active';
        ELSE
            L_Event.Event_Text :=
                'Water runtime healthy';
        END_IF;

        GVL_Water_Runtime_Hardening.G_Event_Log[L_i] :=
            L_Event;

    END_IF;

    L_Any_Rollback :=
        L_Any_Rollback
        OR L_FSM.Rollback_Required;

    L_Any_Escalation :=
        L_Any_Escalation
        OR L_FSM.Escalation_Required;

END_FOR;

GVL_Water_Runtime_Hardening.G_Runtime_Quarantine_Active :=
    L_Any_Escalation;

GVL_Water_Runtime_Hardening.G_Service_Mode_Active := FALSE;
GVL_Water_Runtime_Hardening.G_Maintenance_Mode_Active := FALSE;

GVL_Water_Runtime_Hardening.G_Any_Rollback_Required :=
    L_Any_Rollback;

GVL_Water_Runtime_Hardening.G_Any_Escalation_Required :=
    L_Any_Escalation;

GVL_Water_Runtime_Hardening.G_Runtime_Valid := TRUE;
GVL_Water_Runtime_Hardening.G_Last_Update_MS := VI_System_Time_MS;

IF L_Any_Escalation THEN
    GVL_Water_Runtime_Hardening.G_Status_Code := 2;
    GVL_Water_Runtime_Hardening.G_Status_Text :=
        'Runtime quarantine escalation active';
ELSIF L_Any_Rollback THEN
    GVL_Water_Runtime_Hardening.G_Status_Code := 1;
    GVL_Water_Runtime_Hardening.G_Status_Text :=
        'Recovery rollback active';
ELSE
    GVL_Water_Runtime_Hardening.G_Status_Code := 0;
    GVL_Water_Runtime_Hardening.G_Status_Text :=
        'Production runtime hardening active';
END_IF;
          
END_FUNCTION_BLOCK

FUNCTION_BLOCK FB_Modbus_RTU_Driver
  VAR_INPUT
    VI_Enable : BOOL;
    VI_Driver_Attached : BOOL;
    VI_System_Time_MS : UDINT;
  END_VAR
  VAR_OUTPUT
    VO_Driver_Online : BOOL;
    VO_Driver_Error : BOOL;
    VO_Driver_Error_Code : WORD;
  END_VAR
  VAR
    L_Request_Active : BOOL;
    L_Last_Sequence : UDINT;
    L_Exchange_In_Progress : BOOL;
    L_Last_Success_MS : UDINT;
    FB_TX_Builder : FB_Modbus_RTU_TX_Builder;
    FB_RX_Parser : FB_Modbus_RTU_RX_Parser;
    FB_Response_Apply : FB_Modbus_Response_Apply;
  END_VAR

            // ======================================================
// MODBUS RTU DRIVER ORCHESTRATION
// ======================================================
// Responsibilities:
//   1. Detect active request.
//   2. Build TX frame.
//   3. Wait for physical RX frame.
//   4. Validate/parse RX frame.
//   5. Apply validated response.
//
// IMPORTANT:
//   Real serial exchange is still external.
//   Concrete RTU/COM implementation must:
//      - send G_TX_Frame
//      - fill G_RX_Frame
//      - set G_RX_Ready
// ======================================================

VO_Driver_Online := FALSE;
VO_Driver_Error := FALSE;
VO_Driver_Error_Code := 0;

GVL_MODBUS_RTU_BRIDGE.G_Driver_Online := FALSE;
GVL_MODBUS_RTU_BRIDGE.G_Driver_Error := FALSE;
GVL_MODBUS_RTU_BRIDGE.G_Driver_Error_Code := 0;

IF NOT VI_Enable THEN

    GVL_MODBUS_RTU_BRIDGE.G_Response_Busy := FALSE;
    GVL_MODBUS_RTU_BRIDGE.G_Response_Done := FALSE;
    GVL_MODBUS_RTU_BRIDGE.G_Response_Error := FALSE;
    GVL_MODBUS_RTU_BRIDGE.G_Response_Error_Code := 0;

    GVL_MODBUS_RTU_FRAME.G_TX_Ready := FALSE;
    GVL_MODBUS_RTU_FRAME.G_RX_Ready := FALSE;

    L_Exchange_In_Progress := FALSE;

    RETURN;
END_IF;

IF NOT VI_Driver_Attached THEN

    VO_Driver_Error := TRUE;
    VO_Driver_Error_Code := 16#0002;

    GVL_MODBUS_RTU_BRIDGE.G_Driver_Error := TRUE;
    GVL_MODBUS_RTU_BRIDGE.G_Driver_Error_Code := VO_Driver_Error_Code;

    IF GVL_MODBUS_RTU_BRIDGE.G_Request_Valid THEN

        GVL_MODBUS_RTU_BRIDGE.G_Response_Busy := FALSE;
        GVL_MODBUS_RTU_BRIDGE.G_Response_Done := FALSE;
        GVL_MODBUS_RTU_BRIDGE.G_Response_Error := TRUE;
        GVL_MODBUS_RTU_BRIDGE.G_Response_Error_Code := VO_Driver_Error_Code;

        GVL_MODBUS_RTU_BRIDGE.G_Response_Sequence :=
            GVL_MODBUS_RTU_BRIDGE.G_Request_Sequence;

        GVL_MODBUS_RTU_BRIDGE.G_Response_Update_MS :=
            VI_System_Time_MS;

    END_IF;

    L_Exchange_In_Progress := FALSE;

    RETURN;
END_IF;

// ======================================================
// REQUEST DETECTION
// ======================================================
L_Request_Active := GVL_MODBUS_RTU_BRIDGE.G_Request_Valid;

IF L_Request_Active THEN

    IF GVL_MODBUS_RTU_BRIDGE.G_Request_Sequence <> L_Last_Sequence THEN

        L_Last_Sequence :=
            GVL_MODBUS_RTU_BRIDGE.G_Request_Sequence;

        L_Exchange_In_Progress := TRUE;

        GVL_MODBUS_RTU_BRIDGE.G_Response_Busy := TRUE;
        GVL_MODBUS_RTU_BRIDGE.G_Response_Done := FALSE;
        GVL_MODBUS_RTU_BRIDGE.G_Response_Error := FALSE;
        GVL_MODBUS_RTU_BRIDGE.G_Response_Error_Code := 0;

        // ==============================================
        // BUILD TX FRAME
        // ==============================================
        FB_TX_Builder(
            VI_Request_Valid := TRUE,
            VI_Slave_ID := GVL_MODBUS_RTU_BRIDGE.G_Request_Slave_ID,
            VI_Function_Code := GVL_MODBUS_RTU_BRIDGE.G_Request_Function_Code,
            VI_Start_Register := GVL_MODBUS_RTU_BRIDGE.G_Request_Start_Register,
            VI_Register_Count := GVL_MODBUS_RTU_BRIDGE.G_Request_Register_Count,
            VI_Write_Value := GVL_MODBUS_RTU_BRIDGE.G_Request_Write_Value
        );

        IF FB_TX_Builder.VO_Error THEN

            GVL_MODBUS_RTU_BRIDGE.G_Response_Busy := FALSE;
            GVL_MODBUS_RTU_BRIDGE.G_Response_Done := FALSE;
            GVL_MODBUS_RTU_BRIDGE.G_Response_Error := TRUE;
            GVL_MODBUS_RTU_BRIDGE.G_Response_Error_Code :=
                FB_TX_Builder.VO_Error_Code;

            GVL_MODBUS_RTU_BRIDGE.G_Response_Sequence :=
                GVL_MODBUS_RTU_BRIDGE.G_Request_Sequence;

            GVL_MODBUS_RTU_BRIDGE.G_Response_Update_MS :=
                VI_System_Time_MS;

            L_Exchange_In_Progress := FALSE;

            RETURN;

        END_IF;

        GVL_MODBUS_RTU_FRAME.G_TX_Frame :=
            FB_TX_Builder.VO_Frame;

        GVL_MODBUS_RTU_FRAME.G_TX_Ready := TRUE;
        GVL_MODBUS_RTU_FRAME.G_Last_TX_MS := VI_System_Time_MS;

    END_IF;

END_IF;

// ======================================================
// RX FRAME AVAILABLE
// ======================================================
IF L_Exchange_In_Progress AND
   GVL_MODBUS_RTU_FRAME.G_RX_Ready THEN

    // ==================================================
    // PARSE RX FRAME
    // ==================================================
    FB_RX_Parser(
        VI_Frame := GVL_MODBUS_RTU_FRAME.G_RX_Frame,
        VI_Expected_Slave_ID :=
            GVL_MODBUS_RTU_BRIDGE.G_Request_Slave_ID,
        VI_Expected_Function :=
            GVL_MODBUS_RTU_BRIDGE.G_Request_Function_Code
    );

    // ==================================================
    // APPLY RESPONSE
    // ==================================================
    FB_Response_Apply(
        VI_Request_Valid := TRUE,
        VI_Request_Index := GVL_MODBUS_RTU_BRIDGE.G_Request_Index,
        VI_Request_Sequence :=
            GVL_MODBUS_RTU_BRIDGE.G_Request_Sequence,
        VI_Parser_Valid := FB_RX_Parser.VO_Valid,
        VI_Parser_Error := FB_RX_Parser.VO_Error,
        VI_Parser_Error_Code := FB_RX_Parser.VO_Error_Code,
        VI_Register_Count := FB_RX_Parser.VO_Register_Count,
        VI_Register_Value := FB_RX_Parser.VO_Register_Value,
        VI_System_Time_MS := VI_System_Time_MS
    );

    IF FB_Response_Apply.VO_Response_Applied THEN

        L_Last_Success_MS := VI_System_Time_MS;

        GVL_MODBUS_RTU_FRAME.G_RX_Ready := FALSE;

        L_Exchange_In_Progress := FALSE;

    END_IF;

END_IF;

// ======================================================
// DRIVER ONLINE STATE
// ======================================================
IF (L_Last_Success_MS > 0) AND
   ((VI_System_Time_MS - L_Last_Success_MS) <
    GVL_CONFIG.G_OpenTherm_Heartbeat_Timeout_MS) THEN

    VO_Driver_Online := TRUE;

    GVL_MODBUS_RTU_BRIDGE.G_Driver_Online := TRUE;

END_IF;

// ======================================================
// CLEAR IDLE BUSY STATE
// ======================================================
IF NOT L_Request_Active THEN

    GVL_MODBUS_RTU_BRIDGE.G_Response_Busy := FALSE;

    L_Exchange_In_Progress := FALSE;

END_IF;
          
END_FUNCTION_BLOCK

FUNCTION_BLOCK FB_Heating_Runtime_State_Publication_Phase
  VAR_INPUT
    VI_Enable : BOOL;
    VI_Zone_Valves : ARRAY[1..GVL_CONSTANTS.C_MAX_HEATING_CIRCUITS] OF BOOL;
    VI_Manifold_Pumps : ARRAY[1..GVL_CONSTANTS.C_MAX_MANIFOLDS] OF BOOL;
    VI_Manifold_Valves : ARRAY[1..GVL_CONSTANTS.C_MAX_MANIFOLDS] OF REAL;
    VI_Boiler_OT_Enable : ARRAY[1..GVL_CONSTANTS.C_MAX_BOILERS] OF BOOL;
    VI_Boiler_OT_Setpoint : ARRAY[1..GVL_CONSTANTS.C_MAX_BOILERS] OF REAL;
    VI_Backup_Circulation_Pump : BOOL;
    VI_Electric_Heater_Enable : BOOL;
    VI_Freeze_Risk_Status : BOOL;
    VI_Manifold_Status : ARRAY[1..GVL_CONSTANTS.C_MAX_MANIFOLDS] OF ST_Manifold_Status;
    VI_Boiler_Status : ARRAY[1..GVL_CONSTANTS.C_MAX_BOILERS] OF ST_Boiler_Status;
    VI_DHW_Heating_Pump : BOOL;
    VI_DHW_Circ_Pump : BOOL;
    VI_DHW_Status : ST_DHW_Status;
  END_VAR
  VAR_OUTPUT
    VO_Executed : BOOL;
    VO_Valid : BOOL;
  END_VAR
  VAR
    L_i : INT;
  END_VAR

            // ==============================================================================
// Heating runtime state publication phase
// Owns publication of finalized runtime outputs into global state/status layers.
// Does NOT calculate heating logic and does NOT mutate outputs.
// ==============================================================================



VO_Executed := FALSE;
VO_Valid := FALSE;

IF NOT VI_Enable THEN
    RETURN;
END_IF;

FOR L_i := 1 TO GVL_CONSTANTS.C_MAX_HEATING_CIRCUITS DO
    GVL_STATE.G_Zone_Valves[L_i] := VI_Zone_Valves[L_i];
END_FOR;

FOR L_i := 1 TO GVL_CONSTANTS.C_MAX_MANIFOLDS DO
    GVL_STATE.G_Manifold_Pumps[L_i] := VI_Manifold_Pumps[L_i];
    GVL_STATE.G_Manifold_Valves[L_i] := VI_Manifold_Valves[L_i];
    GVL_STATUS.G_Manifold_Status[L_i] := VI_Manifold_Status[L_i];
END_FOR;

FOR L_i := 1 TO GVL_CONSTANTS.C_MAX_BOILERS DO
    GVL_STATE.G_Boiler_OT_Enable[L_i] := VI_Boiler_OT_Enable[L_i];
    GVL_STATE.G_Boiler_OT_Setpoint[L_i] := VI_Boiler_OT_Setpoint[L_i];
    GVL_STATUS.G_Boiler_Status[L_i] := VI_Boiler_Status[L_i];
END_FOR;

GVL_STATE.G_Backup_Circulation_Pump := VI_Backup_Circulation_Pump;
GVL_STATE.G_Electric_Heater_Enable := VI_Electric_Heater_Enable;
GVL_STATE.G_Safety_Freeze_Risk := VI_Freeze_Risk_Status;
GVL_STATE.G_DHW_Heating_Pump := VI_DHW_Heating_Pump;
GVL_STATE.G_DHW_Circ_Pump := VI_DHW_Circ_Pump;
GVL_STATUS.G_DHW_Status := VI_DHW_Status;

VO_Executed := TRUE;
VO_Valid := TRUE;

// >>> BULK_SYNC_ANCHOR: FB_Heating_Runtime_State_Publication_Phase <<<
          
END_FUNCTION_BLOCK

FUNCTION_BLOCK FB_Trace_Write
  VAR_INPUT
    iLayer : E_Trace_Layer;
    iSource : E_Trace_Source;
    iReason : E_System_Reason_Code;
    iValueBool : BOOL;
    iValueReal : REAL;
    iText : STRING(120);
  END_VAR
  VAR
    L_Index : INT;
  END_VAR

            IF NOT GVL_TRACE.G_Trace_Enabled THEN RETURN; END_IF;

L_Index := GVL_TRACE.G_Trace_Write_Index;

GVL_TRACE.G_Trace_Buffer[L_Index].Timestamp_MS := GVL_TIME_SERVICE.G_Now_MS;
GVL_TRACE.G_Trace_Buffer[L_Index].Layer := iLayer;
GVL_TRACE.G_Trace_Buffer[L_Index].Source := iSource;
GVL_TRACE.G_Trace_Buffer[L_Index].Reason_Code := iReason;
GVL_TRACE.G_Trace_Buffer[L_Index].Value_Bool := iValueBool;
GVL_TRACE.G_Trace_Buffer[L_Index].Value_Real := iValueReal;
GVL_TRACE.G_Trace_Buffer[L_Index].Text := iText;

L_Index := L_Index + 1;
IF L_Index > 200 THEN L_Index := 1; END_IF;

GVL_TRACE.G_Trace_Write_Index := L_Index;
          
END_FUNCTION_BLOCK

FUNCTION_BLOCK FB_Heating_Runtime_Predictive_Correlation_Weighting_Engine
  VAR_INPUT
    VI_Enable : BOOL;
    VI_Runtime_Risk : UINT;
    VI_Cascade_Risk : UINT;
    VI_OT_Risk : UINT;
  END_VAR
  VAR_OUTPUT
    VO_Correlation_Score : UINT;
    VO_Correlation_Degraded : BOOL;
    VO_Status_Code : UINT;
    VO_Status_Text : STRING(128);
  END_VAR
  VAR
    L_Total : UDINT;
  END_VAR

            // ==============================================================================
// Heating runtime predictive correlation weighting engine
// Read-only predictive adaptive correlation layer.
// ==============================================================================



VO_Correlation_Score := 0;
VO_Correlation_Degraded := FALSE;

VO_Status_Code := 0;
VO_Status_Text := 'Heating predictive correlation engine disabled';

IF NOT VI_Enable THEN
    RETURN;
END_IF;

// ======================================================
// SAFE ARITHMETIC
// ======================================================
L_Total :=
    TO_UDINT(VI_Runtime_Risk) +
    TO_UDINT(VI_Cascade_Risk) +
    TO_UDINT(VI_OT_Risk);

VO_Correlation_Score :=
    TO_UINT(L_Total / 3);

// ======================================================
// CORRELATION ANALYSIS
// ======================================================
IF VO_Correlation_Score > 70 THEN
    VO_Correlation_Degraded := TRUE;

    VO_Status_Code := 900;
    VO_Status_Text := 'Heating predictive correlation critical';

ELSIF VO_Correlation_Score > 40 THEN
    VO_Correlation_Degraded := TRUE;

    VO_Status_Code := 200;
    VO_Status_Text := 'Heating predictive correlation degraded';

ELSE
    VO_Status_Code := 1;
    VO_Status_Text := 'Heating predictive correlation nominal';
END_IF;

// >>> BULK_SYNC_ANCHOR: FB_Heating_Runtime_Predictive_Correlation_Weighting_Engine <<<
          
END_FUNCTION_BLOCK

FUNCTION_BLOCK FB_Alarm_Manager
  VAR_INPUT
    VI_System_Time_MS : UDINT;
    VI_IsActivePLC : BOOL;
    VI_Gas_Alarm : BOOL;
    VI_Fire_Alarm : BOOL;
    VI_Flood_Alarm : BOOL;
    VI_Security_Alarm : BOOL;
    VI_First_Fault_Active : BOOL;
    VI_First_Fault_Type : INT;
    VI_First_Fault_Source : INT;
    VI_Security_Msg : STRING(200);
    VI_Acknowledge_All : BOOL;
    VI_Mute_Siren : BOOL;
  END_VAR
  VAR_OUTPUT
    VO_Global_Critical : BOOL;
    VO_Global_Warning : BOOL;
    VO_Siren_Active : BOOL;
    VO_Active_Count : INT;
    VO_Unacked_Count : INT;
    VO_Event_Pulse : BOOL;
    VO_Event_Code : UDINT;
    VO_Event_Value : REAL;
    VO_Alarm_List : ARRAY[1..GVL_CONSTANTS.C_MAX_ALARMS] OF ST_Alarm_Record;
  END_VAR
  VAR_IN_OUT
    VI_Boiler_Errors : ARRAY[1..GVL_CONSTANTS.C_MAX_BOILERS] OF BOOL;
  END_VAR
  VAR_IN_OUT
    VIO_Next_Alarm_ID : UDINT;
  END_VAR
  VAR
    L_i, L_j, L_k : INT;
    L_Target_Slot : INT;
    L_Min_Pri : INT;
    L_Pending_Alarms : ARRAY[1..10] OF ST_Alarm_Record;
    L_Pending_Count : INT := 0;
    T_Debounce_Gas : FB_System_Timer;
    T_Debounce_Fire : FB_System_Timer;
    T_Debounce_Flood : FB_System_Timer;
    T_Debounce_Security : FB_System_Timer;
    R_Trig_Gas : R_TRIG;
    R_Trig_Fire : R_TRIG;
    R_Trig_Flood : R_TRIG;
    R_Trig_Security : R_TRIG;
    R_Trig_First_Fault : R_TRIG;
    R_Trig_Boiler : ARRAY[1..GVL_CONSTANTS.C_MAX_BOILERS] OF R_TRIG;
    L_First_Fault_Source_Text : STRING(32);
    L_First_Fault_Type_Text : STRING(32);
    L_Event_Pulse_Latched : BOOL;
  END_VAR

            VO_Event_Pulse := FALSE;
VO_Event_Code := 0;
VO_Event_Value := 0.0;

// 1. Детекция новых тревог (антидребезг + передний фронт)
T_Debounce_Gas(IN := VI_Gas_Alarm, PT := T#100ms, VI_System_Time_MS := VI_System_Time_MS);
T_Debounce_Fire(IN := VI_Fire_Alarm, PT := T#100ms, VI_System_Time_MS := VI_System_Time_MS);
T_Debounce_Flood(IN := VI_Flood_Alarm, PT := T#500ms, VI_System_Time_MS := VI_System_Time_MS);
T_Debounce_Security(IN := VI_Security_Alarm, PT := T#100ms, VI_System_Time_MS := VI_System_Time_MS);

R_Trig_Gas(CLK := T_Debounce_Gas.Q);
R_Trig_Fire(CLK := T_Debounce_Fire.Q);
R_Trig_Flood(CLK := T_Debounce_Flood.Q);
R_Trig_Security(CLK := T_Debounce_Security.Q);
R_Trig_First_Fault(CLK := VI_First_Fault_Active);
FOR L_i := 1 TO GVL_CONSTANTS.C_MAX_BOILERS DO
    R_Trig_Boiler[L_i](CLK := VI_Boiler_Errors[L_i]);
END_FOR;

// 2. Добавление новых тревог в список (Кольцевой буфер)
L_Pending_Count := 0;
L_Event_Pulse_Latched := FALSE;

IF R_Trig_Gas.Q AND L_Pending_Count < 10 THEN
    L_Pending_Count := L_Pending_Count + 1;
    L_Pending_Alarms[L_Pending_Count].Timestamp_MS := VI_System_Time_MS;
    L_Pending_Alarms[L_Pending_Count].Source := 'Gas';
    L_Pending_Alarms[L_Pending_Count].Source_ID := 0;
    L_Pending_Alarms[L_Pending_Count].Message := 'Критическая концентрация газа!';
    L_Pending_Alarms[L_Pending_Count].Severity := E_ALERT_PRIORITY.ALERT_PRIORITY_CRITICAL;
    L_Pending_Alarms[L_Pending_Count].Is_Active := TRUE;
    L_Pending_Alarms[L_Pending_Count].Is_Acknowledged := FALSE;
END_IF;

IF R_Trig_Fire.Q AND L_Pending_Count < 10 THEN
    L_Pending_Count := L_Pending_Count + 1;
    L_Pending_Alarms[L_Pending_Count].Timestamp_MS := VI_System_Time_MS;
    L_Pending_Alarms[L_Pending_Count].Source := 'Fire';
    L_Pending_Alarms[L_Pending_Count].Source_ID := 0;
    L_Pending_Alarms[L_Pending_Count].Message := 'Обнаружено задымление!';
    L_Pending_Alarms[L_Pending_Count].Severity := E_ALERT_PRIORITY.ALERT_PRIORITY_CRITICAL;
    L_Pending_Alarms[L_Pending_Count].Is_Active := TRUE;
    L_Pending_Alarms[L_Pending_Count].Is_Acknowledged := FALSE;
END_IF;

IF R_Trig_Flood.Q AND L_Pending_Count < 10 THEN
    L_Pending_Count := L_Pending_Count + 1;
    L_Pending_Alarms[L_Pending_Count].Timestamp_MS := VI_System_Time_MS;
    L_Pending_Alarms[L_Pending_Count].Source := 'Flood';
    L_Pending_Alarms[L_Pending_Count].Source_ID := 0;
    L_Pending_Alarms[L_Pending_Count].Message := 'Обнаружена протечка воды!';
    L_Pending_Alarms[L_Pending_Count].Severity := E_ALERT_PRIORITY.ALERT_PRIORITY_CRITICAL;
    L_Pending_Alarms[L_Pending_Count].Is_Active := TRUE;
    L_Pending_Alarms[L_Pending_Count].Is_Acknowledged := FALSE;
END_IF;

IF R_Trig_Security.Q AND L_Pending_Count < 10 THEN
    L_Pending_Count := L_Pending_Count + 1;
    L_Pending_Alarms[L_Pending_Count].Timestamp_MS := VI_System_Time_MS;
    L_Pending_Alarms[L_Pending_Count].Source := 'Security';
    L_Pending_Alarms[L_Pending_Count].Source_ID := 0;
    L_Pending_Alarms[L_Pending_Count].Message := VI_Security_Msg;
    L_Pending_Alarms[L_Pending_Count].Severity := E_ALERT_PRIORITY.ALERT_PRIORITY_CRITICAL;
    L_Pending_Alarms[L_Pending_Count].Is_Active := TRUE;
    L_Pending_Alarms[L_Pending_Count].Is_Acknowledged := FALSE;
END_IF;

IF R_Trig_First_Fault.Q AND L_Pending_Count < 10 THEN
    L_Pending_Count := L_Pending_Count + 1;
    L_Pending_Alarms[L_Pending_Count].Timestamp_MS := VI_System_Time_MS;
    L_Pending_Alarms[L_Pending_Count].Source := 'Diagnostics';
    L_Pending_Alarms[L_Pending_Count].Source_ID := TO_BYTE(VI_First_Fault_Source);

    CASE VI_First_Fault_Type OF
        1: L_First_Fault_Type_Text := 'IO';
        2: L_First_Fault_Type_Text := 'Sensor';
        3: L_First_Fault_Type_Text := 'Comm';
        4: L_First_Fault_Type_Text := 'Subsystem';
        ELSE L_First_Fault_Type_Text := 'Unknown';
    END_CASE;

